LIN {X 0,Y 720.974,Z 317.138,A -85,B 0,C 180,E1 32718.045,E2 32718.045} C_VEL
LIN {X 0,Y 720.181,Z 314.525,A -85,B 0,C 180,E1 32717.982,E2 32717.982} C_VEL
LIN {X 0,Y 720.227,Z 314.61,A -85,B 0,C 180,E1 32716.261,E2 32716.261} C_VEL
LIN {X 0,Y 721.482,Z 317.961,A -85,B 0,C 180,E1 32715.916,E2 32715.916} C_VEL
LIN {X 0,Y 727.5,Z 330.946,A -85,B 0,C 180,E1 32714.519,E2 32714.519} C_VEL
LIN {X 0,Y 727.216,Z 351.094,A -85,B 0,C 180,E1 32713.184,E2 32713.184} C_VEL
LIN {X 0,Y 729.916,Z 362.068,A -85,B 0,C 180,E1 32712.841,E2 32712.841} C_VEL
LIN {X 0,Y 728.769,Z 574.456,A -85,B 0,C 180,E1 32710.185,E2 32710.185} C_VEL
LIN {X 0,Y 727.655,Z 798.892,A -85,B 0,C 180,E1 32707.472,E2 32707.472} C_VEL
LIN {X 0,Y 727.389,Z 834.661,A -85,B 0,C 180,E1 32707.008,E2 32707.008} C_VEL
LIN {X 0,Y 726.992,Z 861.421,A -85,B 0,C 180,E1 32706.503,E2 32706.503} C_VEL
LIN {X 0,Y 726.546,Z 887.78,A -85,B 0,C 180,E1 32705.847,E2 32705.847} C_VEL
LIN {X 0,Y 725.988,Z 915.933,A -85,B 0,C 180,E1 32704.967,E2 32704.967} C_VEL
LIN {X 0,Y 725.356,Z 940.667,A -85,B 0,C 180,E1 32704.031,E2 32704.031} C_VEL
LIN {X 0,Y 724.823,Z 961.723,A -85,B 0,C 180,E1 32703.11,E2 32703.11} C_VEL
LIN {X 0,Y 724.247,Z 986.24,A -85,B 0,C 180,E1 32701.889,E2 32701.889} C_VEL
LIN {X 0,Y 723.55,Z 1010.091,A -85,B 0,C 180,E1 32700.519,E2 32700.519} C_VEL
LIN {X 0,Y 723.012,Z 1029.596,A -85,B 0,C 180,E1 32699.265,E2 32699.265} C_VEL
LIN {X 0,Y 722.479,Z 1051.277,A -85,B 0,C 180,E1 32697.71,E2 32697.71} C_VEL
LIN {X 0,Y 721.914,Z 1071.822,A -85,B 0,C 180,E1 32696.043,E2 32696.043} C_VEL
LIN {X 0,Y 721.493,Z 1089.789,A -85,B 0,C 180,E1 32694.423,E2 32694.423} C_VEL
LIN {X 0,Y 721.059,Z 1108.723,A -85,B 0,C 180,E1 32692.501,E2 32692.501} C_VEL
LIN {X 0,Y 720.779,Z 1122.974,A -85,B 0,C 180,E1 32690.885,E2 32690.885} C_VEL
LIN {X 0,Y 720.524,Z 1137.042,A -85,B 0,C 180,E1 32689.116,E2 32689.116} C_VEL
LIN {X 0,Y 720.309,Z 1152.141,A -85,B 0,C 180,E1 32686.947,E2 32686.947} C_VEL
LIN {X 0,Y 720.143,Z 1162.707,A -85,B 0,C 180,E1 32685.207,E2 32685.207} C_VEL
LIN {X 0,Y 720.071,Z 1171.491,A -85,B 0,C 180,E1 32683.571,E2 32683.571} C_VEL
LIN {X 0,Y 719.987,Z 1179.518,A -85,B 0,C 180,E1 32681.86,E2 32681.86} C_VEL
LIN {X 0,Y 719.96,Z 1187.317,A -85,B 0,C 180,E1 32679.915,E2 32679.915} C_VEL
LIN {X 0,Y 719.934,Z 1194.039,A -85,B 0,C 180,E1 32677.822,E2 32677.822} C_VEL
LIN {X 0,Y 719.92,Z 1199.281,A -85,B 0,C 180,E1 32675.658,E2 32675.658} C_VEL
LIN {X 0,Y 719.915,Z 1202.793,A -85,B 0,C 180,E1 32673.503,E2 32673.503} C_VEL
LIN {X 0,Y 719.914,Z 1204.613,A -85,B 0,C 180,E1 32671.432,E2 32671.432} C_VEL
LIN {X 0,Y 719.891,Z 1204.859,A -85,B 0,C 180,E1 32669.442,E2 32669.442} C_VEL
LIN {X 0,Y 719.906,Z 1203.907,A -85,B 0,C 180,E1 32667.531,E2 32667.531} C_VEL
LIN {X 0,Y 719.907,Z 1201.173,A -85,B 0,C 180,E1 32665.379,E2 32665.379} C_VEL
LIN {X 0,Y 719.917,Z 1196.95,A -85,B 0,C 180,E1 32663.299,E2 32663.299} C_VEL
LIN {X 0,Y 719.939,Z 1191.157,A -85,B 0,C 180,E1 32661.211,E2 32661.211} C_VEL
LIN {X 0,Y 719.966,Z 1183.315,A -85,B 0,C 180,E1 32659.031,E2 32659.031} C_VEL
LIN {X 0,Y 720.059,Z 1173.533,A -85,B 0,C 180,E1 32656.836,E2 32656.836} C_VEL
LIN {X 0,Y 720.129,Z 1164.06,A -85,B 0,C 180,E1 32655.032,E2 32655.032} C_VEL
LIN {X 0,Y 720.263,Z 1154.218,A -85,B 0,C 180,E1 32653.382,E2 32653.382} C_VEL
LIN {X 0,Y 720.451,Z 1141.93,A -85,B 0,C 180,E1 32651.552,E2 32651.552} C_VEL
LIN {X 0,Y 720.732,Z 1125.799,A -85,B 0,C 180,E1 32649.451,E2 32649.451} C_VEL
LIN {X 0,Y 720.989,Z 1111.824,A -85,B 0,C 180,E1 32647.838,E2 32647.838} C_VEL
LIN {X 0,Y 721.308,Z 1097.116,A -85,B 0,C 180,E1 32646.296,E2 32646.296} C_VEL
LIN {X 0,Y 721.786,Z 1077.871,A -85,B 0,C 180,E1 32644.479,E2 32644.479} C_VEL
LIN {X 0,Y 722.256,Z 1058.515,A -85,B 0,C 180,E1 32642.86,E2 32642.86} C_VEL
LIN {X 0,Y 722.862,Z 1037.525,A -85,B 0,C 180,E1 32641.28,E2 32641.28} C_VEL
LIN {X 0,Y 723.411,Z 1014.532,A -85,B 0,C 180,E1 32639.754,E2 32639.754} C_VEL
LIN {X 0,Y 723.994,Z 993.832,A -85,B 0,C 180,E1 32638.53,E2 32638.53} C_VEL
LIN {X 0,Y 724.698,Z 969.545,A -85,B 0,C 180,E1 32637.258,E2 32637.258} C_VEL
LIN {X 0,Y 725.281,Z 944.345,A -85,B 0,C 180,E1 32636.122,E2 32636.122} C_VEL
LIN {X 0,Y 725.805,Z 921.337,A -85,B 0,C 180,E1 32635.226,E2 32635.226} C_VEL
LIN {X 0,Y 726.415,Z 895.267,A -85,B 0,C 180,E1 32634.366,E2 32634.366} C_VEL
LIN {X 0,Y 726.881,Z 868.856,A -85,B 0,C 180,E1 32633.665,E2 32633.665} C_VEL
LIN {X 0,Y 727.285,Z 842.382,A -85,B 0,C 180,E1 32633.122,E2 32633.122} C_VEL
LIN {X 0,Y 727.575,Z 814.613,A -85,B 0,C 180,E1 32632.715,E2 32632.715} C_VEL
LIN {X 0,Y 728.684,Z 590.147,A -85,B 0,C 180,E1 32630.008,E2 32630.008} C_VEL
LIN {X 0,Y 729.786,Z 383.764,A -85,B 0,C 180,E1 32627.434,E2 32627.434} C_VEL
LIN {X 0,Y 729.82,Z 346.15,A -85,B 0,C 180,E1 32626.943,E2 32626.943} C_VEL
LIN {X 0,Y 729.774,Z 330.048,A -85,B 0,C 180,E1 32626.614,E2 32626.614} C_VEL
LIN {X 0,Y 725.417,Z 323.688,A -85,B 0,C 180,E1 32626.156,E2 32626.156} C_VEL
LIN {X 0,Y 722.735,Z 319.452,A -85,B 0,C 180,E1 32625.864,E2 32625.864} C_VEL
LIN {X 0,Y 720.686,Z 316.455,A -85,B 0,C 180,E1 32625.642,E2 32625.642} C_VEL
LIN {X 0,Y 720.203,Z 314.522,A -85,B 0,C 180,E1 32625.545,E2 32625.545} C_VEL
LIN {X 0,Y 720.215,Z 314.522,A -85,B 0,C 180,E1 32622.624,E2 32622.624} C_VEL
LIN {X 0,Y 720.181,Z 314.519,A -85,B 0,C 180,E1 32619.692,E2 32619.692} C_VEL
LIN {X 0,Y 720.194,Z 314.503,A -85,B 0,C 180,E1 32616.854,E2 32616.854} C_VEL
LIN {X 0,Y 720.217,Z 314.522,A -85,B 0,C 180,E1 32613.879,E2 32613.879} C_VEL
LIN {X 0,Y 720.207,Z 314.506,A -85,B 0,C 180,E1 32610.908,E2 32610.908} C_VEL
LIN {X 0,Y 720.201,Z 314.521,A -85,B 0,C 180,E1 32607.807,E2 32607.807} C_VEL
LIN {X 0,Y 720.208,Z 314.502,A -85,B 0,C 180,E1 32604.877,E2 32604.877} C_VEL
LIN {X 0,Y 720.204,Z 314.521,A -85,B 0,C 180,E1 32601.93,E2 32601.93} C_VEL
LIN {X 0,Y 720.18,Z 314.522,A -85,B 0,C 180,E1 32599.043,E2 32599.043} C_VEL
LIN {X 0,Y 720.208,Z 314.518,A -85,B 0,C 180,E1 32596.11,E2 32596.11} C_VEL
LIN {X 0,Y 720.218,Z 314.522,A -85,B 0,C 180,E1 32593.161,E2 32593.161} C_VEL
LIN {X 0,Y 720.218,Z 314.767,A -85,B 0,C 180,E1 32591.228,E2 32591.228} C_VEL
LIN {X 0,Y 721.001,Z 318.867,A -85,B 0,C 180,E1 32591.074,E2 32591.074} C_VEL
LIN {X 0,Y 721.049,Z 390.816,A -85,B 0,C 180,E1 32588.611,E2 32588.611} C_VEL
LIN {X 0,Y 721.392,Z 472.664,A -85,B 0,C 180,E1 32585.688,E2 32585.688} C_VEL
LIN {X 0,Y 721.652,Z 538.695,A -85,B 0,C 180,E1 32583.257,E2 32583.257} C_VEL
LIN {X 0,Y 721.594,Z 602.053,A -85,B 0,C 180,E1 32580.873,E2 32580.873} C_VEL
LIN {X 0,Y 721.303,Z 676.449,A -85,B 0,C 180,E1 32578.054,E2 32578.054} C_VEL
LIN {X 0,Y 720.86,Z 755.637,A -85,B 0,C 180,E1 32575.027,E2 32575.027} C_VEL
LIN {X 0,Y 720.503,Z 836.2,A -85,B 0,C 180,E1 32571.989,E2 32571.989} C_VEL
LIN {X 0,Y 720.594,Z 839.219,A -85,B 0,C 180,E1 32571.958,E2 32571.958} C_VEL
LIN {X 0,Y 719.614,Z 846.884,A -85,B 0,C 180,E1 32571.896,E2 32571.896} C_VEL
LIN {X 0,Y 713.449,Z 867.175,A -85,B 0,C 180,E1 32571.788,E2 32571.788} C_VEL
LIN {X 0,Y 712.686,Z 873.758,A -85,B 0,C 180,E1 32571.734,E2 32571.734} C_VEL
LIN {X 0,Y 712.588,Z 952.533,A -85,B 0,C 180,E1 32570.922,E2 32570.922} C_VEL
LIN {X 0,Y 712.499,Z 966.842,A -85,B 0,C 180,E1 32570.631,E2 32570.631} C_VEL
LIN {X 0,Y 712.403,Z 980.206,A -85,B 0,C 180,E1 32570.222,E2 32570.222} C_VEL
LIN {X 0,Y 712.317,Z 993.078,A -85,B 0,C 180,E1 32569.69,E2 32569.69} C_VEL
LIN {X 0,Y 712.198,Z 1005.778,A -85,B 0,C 180,E1 32568.992,E2 32568.992} C_VEL
LIN {X 0,Y 712.115,Z 1016.953,A -85,B 0,C 180,E1 32568.212,E2 32568.212} C_VEL
LIN {X 0,Y 712.032,Z 1027.591,A -85,B 0,C 180,E1 32567.263,E2 32567.263} C_VEL
LIN {X 0,Y 711.981,Z 1035.549,A -85,B 0,C 180,E1 32566.353,E2 32566.353} C_VEL
LIN {X 0,Y 711.939,Z 1042.963,A -85,B 0,C 180,E1 32565.273,E2 32565.273} C_VEL
LIN {X 0,Y 711.925,Z 1048.677,A -85,B 0,C 180,E1 32564.105,E2 32564.105} C_VEL
LIN {X 0,Y 711.914,Z 1052.056,A -85,B 0,C 180,E1 32563.098,E2 32563.098} C_VEL
LIN {X 0,Y 711.918,Z 1054.136,A -85,B 0,C 180,E1 32562.086,E2 32562.086} C_VEL
LIN {X 0,Y 711.912,Z 1054.947,A -85,B 0,C 180,E1 32560.813,E2 32560.813} C_VEL
LIN {X 0,Y 711.918,Z 1053.936,A -85,B 0,C 180,E1 32559.701,E2 32559.701} C_VEL
LIN {X 0,Y 711.913,Z 1051.897,A -85,B 0,C 180,E1 32558.754,E2 32558.754} C_VEL
LIN {X 0,Y 711.926,Z 1048.316,A -85,B 0,C 180,E1 32557.715,E2 32557.715} C_VEL
LIN {X 0,Y 711.943,Z 1042.145,A -85,B 0,C 180,E1 32556.507,E2 32556.507} C_VEL
LIN {X 0,Y 711.982,Z 1035.188,A -85,B 0,C 180,E1 32555.511,E2 32555.511} C_VEL
LIN {X 0,Y 712.041,Z 1026.599,A -85,B 0,C 180,E1 32554.547,E2 32554.547} C_VEL
LIN {X 0,Y 712.12,Z 1016.444,A -85,B 0,C 180,E1 32553.66,E2 32553.66} C_VEL
LIN {X 0,Y 712.195,Z 1006.167,A -85,B 0,C 180,E1 32552.943,E2 32552.943} C_VEL
LIN {X 0,Y 712.308,Z 994.071,A -85,B 0,C 180,E1 32552.268,E2 32552.268} C_VEL
LIN {X 0,Y 712.4,Z 980.752,A -85,B 0,C 180,E1 32551.707,E2 32551.707} C_VEL
LIN {X 0,Y 712.484,Z 968.261,A -85,B 0,C 180,E1 32551.317,E2 32551.317} C_VEL
LIN {X 0,Y 712.585,Z 953.301,A -85,B 0,C 180,E1 32550.998,E2 32550.998} C_VEL
LIN {X 0,Y 712.639,Z 907.094,A -85,B 0,C 180,E1 32550.51,E2 32550.51} C_VEL
LIN {X 0,Y 712.62,Z 835.481,A -85,B 0,C 180,E1 32549.777,E2 32549.777} C_VEL
LIN {X 0,Y 713.066,Z 754.769,A -85,B 0,C 180,E1 32546.693,E2 32546.693} C_VEL
LIN {X 0,Y 713.49,Z 681.049,A -85,B 0,C 180,E1 32543.871,E2 32543.871} C_VEL
LIN {X 0,Y 713.925,Z 601.874,A -85,B 0,C 180,E1 32540.828,E2 32540.828} C_VEL
LIN {X 0,Y 714.318,Z 528.018,A -85,B 0,C 180,E1 32537.948,E2 32537.948} C_VEL
LIN {X 0,Y 714.295,Z 457.43,A -85,B 0,C 180,E1 32535.27,E2 32535.27} C_VEL
LIN {X 0,Y 714.435,Z 399.388,A -85,B 0,C 180,E1 32533.044,E2 32533.044} C_VEL
LIN {X 0,Y 715.772,Z 401.418,A -85,B 0,C 180,E1 32532.916,E2 32532.916} C_VEL
LIN {X 0,Y 717.784,Z 401.457,A -85,B 0,C 180,E1 32532.766,E2 32532.766} C_VEL
LIN {X 0,Y 720.642,Z 399.11,A -85,B 0,C 180,E1 32532.587,E2 32532.587} C_VEL
LIN {X 0,Y 723.62,Z 394.867,A -85,B 0,C 180,E1 32532.427,E2 32532.427} C_VEL
LIN {X 0,Y 722.239,Z 609.654,A -85,B 0,C 180,E1 32529.747,E2 32529.747} C_VEL
LIN {X 0,Y 721.025,Z 799.484,A -85,B 0,C 180,E1 32527.427,E2 32527.427} C_VEL
LIN {X 0,Y 720.629,Z 826.478,A -85,B 0,C 180,E1 32526.947,E2 32526.947} C_VEL
LIN {X 0,Y 720.054,Z 853.632,A -85,B 0,C 180,E1 32526.296,E2 32526.296} C_VEL
LIN {X 0,Y 719.485,Z 877.07,A -85,B 0,C 180,E1 32525.591,E2 32525.591} C_VEL
LIN {X 0,Y 718.87,Z 901.756,A -85,B 0,C 180,E1 32524.711,E2 32524.711} C_VEL
LIN {X 0,Y 718.073,Z 927.462,A -85,B 0,C 180,E1 32523.623,E2 32523.623} C_VEL
LIN {X 0,Y 717.352,Z 949.468,A -85,B 0,C 180,E1 32522.55,E2 32522.55} C_VEL
LIN {X 0,Y 716.647,Z 971.848,A -85,B 0,C 180,E1 32521.314,E2 32521.314} C_VEL
LIN {X 0,Y 715.878,Z 995.614,A -85,B 0,C 180,E1 32519.818,E2 32519.818} C_VEL
LIN {X 0,Y 715.153,Z 1017.098,A -85,B 0,C 180,E1 32518.293,E2 32518.293} C_VEL
LIN {X 0,Y 714.487,Z 1039.264,A -85,B 0,C 180,E1 32516.515,E2 32516.515} C_VEL
LIN {X 0,Y 713.89,Z 1057.779,A -85,B 0,C 180,E1 32514.847,E2 32514.847} C_VEL
LIN {X 0,Y 713.401,Z 1076.74,A -85,B 0,C 180,E1 32512.933,E2 32512.933} C_VEL
LIN {X 0,Y 713.009,Z 1091.871,A -85,B 0,C 180,E1 32511.212,E2 32511.212} C_VEL
LIN {X 0,Y 712.716,Z 1104.738,A -85,B 0,C 180,E1 32509.592,E2 32509.592} C_VEL
LIN {X 0,Y 712.476,Z 1116.839,A -85,B 0,C 180,E1 32507.9,E2 32507.9} C_VEL
LIN {X 0,Y 712.266,Z 1130.542,A -85,B 0,C 180,E1 32505.721,E2 32505.721} C_VEL
LIN {X 0,Y 712.109,Z 1140.422,A -85,B 0,C 180,E1 32503.894,E2 32503.894} C_VEL
LIN {X 0,Y 712.02,Z 1148.589,A -85,B 0,C 180,E1 32502.161,E2 32502.161} C_VEL
LIN {X 0,Y 711.984,Z 1156.257,A -85,B 0,C 180,E1 32500.275,E2 32500.275} C_VEL
LIN {X 0,Y 711.941,Z 1163.451,A -85,B 0,C 180,E1 32498.075,E2 32498.075} C_VEL
LIN {X 0,Y 711.921,Z 1169.015,A -85,B 0,C 180,E1 32495.805,E2 32495.805} C_VEL
LIN {X 0,Y 711.911,Z 1172.518,A -85,B 0,C 180,E1 32493.705,E2 32493.705} C_VEL
LIN {X 0,Y 711.907,Z 1174.501,A -85,B 0,C 180,E1 32491.611,E2 32491.611} C_VEL
LIN {X 0,Y 711.891,Z 1174.879,A -85,B 0,C 180,E1 32489.438,E2 32489.438} C_VEL
LIN {X 0,Y 711.906,Z 1173.876,A -85,B 0,C 180,E1 32487.425,E2 32487.425} C_VEL
LIN {X 0,Y 711.912,Z 1170.996,A -85,B 0,C 180,E1 32485.167,E2 32485.167} C_VEL
LIN {X 0,Y 711.918,Z 1166.663,A -85,B 0,C 180,E1 32483.064,E2 32483.064} C_VEL
LIN {X 0,Y 711.945,Z 1161.033,A -85,B 0,C 180,E1 32481.033,E2 32481.033} C_VEL
LIN {X 0,Y 711.994,Z 1153.18,A -85,B 0,C 180,E1 32478.827,E2 32478.827} C_VEL
LIN {X 0,Y 712.092,Z 1143.342,A -85,B 0,C 180,E1 32476.605,E2 32476.605} C_VEL
LIN {X 0,Y 712.179,Z 1134.313,A -85,B 0,C 180,E1 32474.863,E2 32474.863} C_VEL
LIN {X 0,Y 712.339,Z 1125.015,A -85,B 0,C 180,E1 32473.278,E2 32473.278} C_VEL
LIN {X 0,Y 712.524,Z 1114.561,A -85,B 0,C 180,E1 32471.68,E2 32471.68} C_VEL
LIN {X 0,Y 712.768,Z 1102.854,A -85,B 0,C 180,E1 32470.07,E2 32470.07} C_VEL
LIN {X 0,Y 713.126,Z 1087.636,A -85,B 0,C 180,E1 32468.189,E2 32468.189} C_VEL
LIN {X 0,Y 713.541,Z 1070.143,A -85,B 0,C 180,E1 32466.287,E2 32466.287} C_VEL
LIN {X 0,Y 714.064,Z 1053.157,A -85,B 0,C 180,E1 32464.63,E2 32464.63} C_VEL
LIN {X 0,Y 714.675,Z 1031.871,A -85,B 0,C 180,E1 32462.776,E2 32462.776} C_VEL
LIN {X 0,Y 715.4,Z 1010.459,A -85,B 0,C 180,E1 32461.127,E2 32461.127} C_VEL
LIN {X 0,Y 716.16,Z 985.918,A -85,B 0,C 180,E1 32459.457,E2 32459.457} C_VEL
LIN {X 0,Y 716.879,Z 964.641,A -85,B 0,C 180,E1 32458.183,E2 32458.183} C_VEL
LIN {X 0,Y 717.707,Z 940.482,A -85,B 0,C 180,E1 32456.9,E2 32456.9} C_VEL
LIN {X 0,Y 718.42,Z 915.161,A -85,B 0,C 180,E1 32455.745,E2 32455.745} C_VEL
LIN {X 0,Y 719.049,Z 892.538,A -85,B 0,C 180,E1 32454.853,E2 32454.853} C_VEL
LIN {X 0,Y 719.738,Z 867.444,A -85,B 0,C 180,E1 32454.012,E2 32454.012} C_VEL
LIN {X 0,Y 720.315,Z 841.314,A -85,B 0,C 180,E1 32453.298,E2 32453.298} C_VEL
LIN {X 0,Y 720.797,Z 815.662,A -85,B 0,C 180,E1 32452.753,E2 32452.753} C_VEL
LIN {X 0,Y 721.142,Z 789.799,A -85,B 0,C 180,E1 32452.349,E2 32452.349} C_VEL
LIN {X 0,Y 722.555,Z 560.025,A -85,B 0,C 180,E1 32449.552,E2 32449.552} C_VEL
LIN {X 0,Y 723.897,Z 350.731,A -85,B 0,C 180,E1 32446.919,E2 32446.919} C_VEL
LIN {X 0,Y 723.883,Z 335.4,A -85,B 0,C 180,E1 32446.714,E2 32446.714} C_VEL
LIN {X 0,Y 714.337,Z 320.821,A -85,B 0,C 180,E1 32445.781,E2 32445.781} C_VEL
LIN {X 0,Y 712.281,Z 315.553,A -85,B 0,C 180,E1 32445.22,E2 32445.22} C_VEL
LIN {X 0,Y 712.261,Z 315.511,A -85,B 0,C 180,E1 32442.287,E2 32442.287} C_VEL
LIN {X 0,Y 712.284,Z 315.51,A -85,B 0,C 180,E1 32439.28,E2 32439.28} C_VEL
LIN {X 0,Y 712.253,Z 315.509,A -85,B 0,C 180,E1 32436.429,E2 32436.429} C_VEL
LIN {X 0,Y 712.28,Z 315.493,A -85,B 0,C 180,E1 32433.387,E2 32433.387} C_VEL
LIN {X 0,Y 712.249,Z 315.508,A -85,B 0,C 180,E1 32430.45,E2 32430.45} C_VEL
LIN {X 0,Y 712.277,Z 315.508,A -85,B 0,C 180,E1 32427.507,E2 32427.507} C_VEL
LIN {X 0,Y 712.248,Z 315.498,A -85,B 0,C 180,E1 32424.541,E2 32424.541} C_VEL
LIN {X 0,Y 712.277,Z 315.507,A -85,B 0,C 180,E1 32421.666,E2 32421.666} C_VEL
LIN {X 0,Y 712.264,Z 315.508,A -85,B 0,C 180,E1 32418.64,E2 32418.64} C_VEL
LIN {X 0,Y 712.278,Z 315.495,A -85,B 0,C 180,E1 32415.72,E2 32415.72} C_VEL
LIN {X 0,Y 712.279,Z 315.508,A -85,B 0,C 180,E1 32412.65,E2 32412.65} C_VEL
LIN {X 0,Y 712.267,Z 315.505,A -85,B 0,C 180,E1 32409.698,E2 32409.698} C_VEL
LIN {X 0,Y 712.284,Z 315.495,A -85,B 0,C 180,E1 32406.529,E2 32406.529} C_VEL
LIN {X 0,Y 712.252,Z 315.511,A -85,B 0,C 180,E1 32403.622,E2 32403.622} C_VEL
LIN {X 0,Y 712.268,Z 315.502,A -85,B 0,C 180,E1 32400.643,E2 32400.643} C_VEL
LIN {X 0,Y 712.251,Z 315.5,A -85,B 0,C 180,E1 32397.747,E2 32397.747} C_VEL
LIN {X 0,Y 712.259,Z 315.512,A -85,B 0,C 180,E1 32394.926,E2 32394.926} C_VEL
LIN {X 0,Y 712.259,Z 315.505,A -85,B 0,C 180,E1 32392.011,E2 32392.011} C_VEL
LIN {X 0,Y 712.257,Z 315.493,A -85,B 0,C 180,E1 32389.075,E2 32389.075} C_VEL
LIN {X 0,Y 712.282,Z 315.496,A -85,B 0,C 180,E1 32386.111,E2 32386.111} C_VEL
LIN {X 0,Y 712.274,Z 315.499,A -85,B 0,C 180,E1 32383.023,E2 32383.023} C_VEL
LIN {X 0,Y 712.271,Z 315.64,A -85,B 0,C 180,E1 32381.358,E2 32381.358} C_VEL
LIN {X 0,Y 713.397,Z 318.736,A -85,B 0,C 180,E1 32380.939,E2 32380.939} C_VEL
LIN {X 0,Y 714.941,Z 320.902,A -85,B 0,C 180,E1 32380.558,E2 32380.558} C_VEL
LIN {X 0,Y 716.779,Z 324.574,A -85,B 0,C 180,E1 32380.015,E2 32380.015} C_VEL
LIN {X 0,Y 722.61,Z 335.701,A -85,B 0,C 180,E1 32378.403,E2 32378.403} C_VEL
LIN {X 0,Y 724.706,Z 339.886,A -85,B 0,C 180,E1 32377.83,E2 32377.83} C_VEL
LIN {X 0,Y 723.691,Z 373.738,A -85,B 0,C 180,E1 32375.251,E2 32375.251} C_VEL
LIN {X 0,Y 722.636,Z 410.919,A -85,B 0,C 180,E1 32372.564,E2 32372.564} C_VEL
LIN {X 0,Y 721.619,Z 447.74,A -85,B 0,C 180,E1 32370.027,E2 32370.027} C_VEL
LIN {X 0,Y 720.698,Z 486.146,A -85,B 0,C 180,E1 32367.483,E2 32367.483} C_VEL
LIN {X 0,Y 720.014,Z 532.442,A -85,B 0,C 180,E1 32364.515,E2 32364.515} C_VEL
LIN {X 0,Y 721.38,Z 542.753,A -85,B 0,C 180,E1 32363.772,E2 32363.772} C_VEL
LIN {X 0,Y 724.081,Z 551.021,A -85,B 0,C 180,E1 32363.08,E2 32363.08} C_VEL
LIN {X 0,Y 728.039,Z 557.601,A -85,B 0,C 180,E1 32362.425,E2 32362.425} C_VEL
LIN {X 0,Y 733.462,Z 562.874,A -85,B 0,C 180,E1 32361.763,E2 32361.763} C_VEL
LIN {X 0,Y 736.609,Z 564.647,A -85,B 0,C 180,E1 32361.305,E2 32361.305} C_VEL
LIN {X 0,Y 738.892,Z 564.846,A -85,B 0,C 180,E1 32360.805,E2 32360.805} C_VEL
LIN {X 0,Y 739.939,Z 563.782,A -85,B 0,C 180,E1 32360.37,E2 32360.37} C_VEL
LIN {X 0,Y 739.975,Z 561.222,A -85,B 0,C 180,E1 32359.887,E2 32359.887} C_VEL
LIN {X 0,Y 738.724,Z 557.439,A -85,B 0,C 180,E1 32359.463,E2 32359.463} C_VEL
LIN {X 0,Y 736.318,Z 552.666,A -85,B 0,C 180,E1 32359.129,E2 32359.129} C_VEL
LIN {X 0,Y 731.678,Z 544.076,A -85,B 0,C 180,E1 32358.795,E2 32358.795} C_VEL
LIN {X 0,Y 727.831,Z 533.761,A -85,B 0,C 180,E1 32358.529,E2 32358.529} C_VEL
LIN {X 0,Y 725.166,Z 522.044,A -85,B 0,C 180,E1 32358.343,E2 32358.343} C_VEL
LIN {X 0,Y 723.697,Z 508.332,A -85,B 0,C 180,E1 32358.239,E2 32358.239} C_VEL
LIN {X 0,Y 723.434,Z 499.656,A -85,B 0,C 180,E1 32358.22,E2 32358.22} C_VEL
LIN {X 0,Y 723.393,Z 331.167,A -85,B 0,C 180,E1 32358.217,E2 32358.217} C_VEL
LIN {X 0,Y 716.339,Z 322.153,A -85,B 0,C 180,E1 32357.711,E2 32357.711} C_VEL
LIN {X 0,Y 715.23,Z 320.781,A -85,B 0,C 180,E1 32357.63,E2 32357.63} C_VEL
LIN {X 0,Y 713.016,Z 317.997,A -85,B 0,C 180,E1 32357.468,E2 32357.468} C_VEL
LIN {X 0,Y 712.282,Z 315.51,A -85,B 0,C 180,E1 32357.413,E2 32357.413} C_VEL
LIN {X 0,Y 712.272,Z 315.647,A -85,B 0,C 180,E1 32356.857,E2 32356.857} C_VEL
LIN {X 0,Y 713.468,Z 318.85,A -85,B 0,C 180,E1 32356.519,E2 32356.519} C_VEL
LIN {X 0,Y 714.541,Z 321.035,A -85,B 0,C 180,E1 32356.268,E2 32356.268} C_VEL
LIN {X 0,Y 721.038,Z 335.061,A -85,B 0,C 180,E1 32354.736,E2 32354.736} C_VEL
LIN {X 0,Y 720.77,Z 351.039,A -85,B 0,C 180,E1 32353.667,E2 32353.667} C_VEL
LIN {X 0,Y 724.023,Z 364.243,A -85,B 0,C 180,E1 32353.246,E2 32353.246} C_VEL
LIN {X 0,Y 722.638,Z 575.911,A -85,B 0,C 180,E1 32350.578,E2 32350.578} C_VEL
LIN {X 0,Y 721.293,Z 799.655,A -85,B 0,C 180,E1 32347.851,E2 32347.851} C_VEL
LIN {X 0,Y 720.976,Z 834.996,A -85,B 0,C 180,E1 32347.388,E2 32347.388} C_VEL
LIN {X 0,Y 720.495,Z 862.1,A -85,B 0,C 180,E1 32346.871,E2 32346.871} C_VEL
LIN {X 0,Y 719.956,Z 888.321,A -85,B 0,C 180,E1 32346.211,E2 32346.211} C_VEL
LIN {X 0,Y 719.275,Z 916.723,A -85,B 0,C 180,E1 32345.312,E2 32345.312} C_VEL
LIN {X 0,Y 718.555,Z 940.783,A -85,B 0,C 180,E1 32344.393,E2 32344.393} C_VEL
LIN {X 0,Y 717.878,Z 962.623,A -85,B 0,C 180,E1 32343.43,E2 32343.43} C_VEL
LIN {X 0,Y 717.154,Z 987.366,A -85,B 0,C 180,E1 32342.18,E2 32342.18} C_VEL
LIN {X 0,Y 716.342,Z 1010.822,A -85,B 0,C 180,E1 32340.813,E2 32340.813} C_VEL
LIN {X 0,Y 715.668,Z 1031.083,A -85,B 0,C 180,E1 32339.492,E2 32339.492} C_VEL
LIN {X 0,Y 714.978,Z 1053.564,A -85,B 0,C 180,E1 32337.844,E2 32337.844} C_VEL
LIN {X 0,Y 714.327,Z 1073.414,A -85,B 0,C 180,E1 32336.2,E2 32336.2} C_VEL
LIN {X 0,Y 713.795,Z 1092.87,A -85,B 0,C 180,E1 32334.407,E2 32334.407} C_VEL
LIN {X 0,Y 713.307,Z 1109.504,A -85,B 0,C 180,E1 32332.672,E2 32332.672} C_VEL
LIN {X 0,Y 712.982,Z 1122.976,A -85,B 0,C 180,E1 32331.124,E2 32331.124} C_VEL
LIN {X 0,Y 712.667,Z 1137.046,A -85,B 0,C 180,E1 32329.335,E2 32329.335} C_VEL
LIN {X 0,Y 712.399,Z 1152.144,A -85,B 0,C 180,E1 32327.141,E2 32327.141} C_VEL
LIN {X 0,Y 712.202,Z 1163.143,A -85,B 0,C 180,E1 32325.303,E2 32325.303} C_VEL
LIN {X 0,Y 712.104,Z 1172.315,A -85,B 0,C 180,E1 32323.56,E2 32323.56} C_VEL
LIN {X 0,Y 712.01,Z 1180.951,A -85,B 0,C 180,E1 32321.666,E2 32321.666} C_VEL
LIN {X 0,Y 711.958,Z 1188.746,A -85,B 0,C 180,E1 32319.62,E2 32319.62} C_VEL
LIN {X 0,Y 711.929,Z 1195.357,A -85,B 0,C 180,E1 32317.423,E2 32317.423} C_VEL
LIN {X 0,Y 711.917,Z 1200.046,A -85,B 0,C 180,E1 32315.318,E2 32315.318} C_VEL
LIN {X 0,Y 711.917,Z 1203.274,A -85,B 0,C 180,E1 32313.139,E2 32313.139} C_VEL
LIN {X 0,Y 711.915,Z 1204.727,A -85,B 0,C 180,E1 32311.045,E2 32311.045} C_VEL
LIN {X 0,Y 711.895,Z 1204.816,A -85,B 0,C 180,E1 32309.275,E2 32309.275} C_VEL
LIN {X 0,Y 711.909,Z 1203.75,A -85,B 0,C 180,E1 32307.342,E2 32307.342} C_VEL
LIN {X 0,Y 711.914,Z 1200.922,A -85,B 0,C 180,E1 32305.165,E2 32305.165} C_VEL
LIN {X 0,Y 711.926,Z 1196.362,A -85,B 0,C 180,E1 32302.981,E2 32302.981} C_VEL
LIN {X 0,Y 711.949,Z 1190.352,A -85,B 0,C 180,E1 32300.868,E2 32300.868} C_VEL
LIN {X 0,Y 712.006,Z 1182.678,A -85,B 0,C 180,E1 32298.743,E2 32298.743} C_VEL
LIN {X 0,Y 712.1,Z 1173.126,A -85,B 0,C 180,E1 32296.603,E2 32296.603} C_VEL
LIN {X 0,Y 712.183,Z 1164.063,A -85,B 0,C 180,E1 32294.862,E2 32294.862} C_VEL
LIN {X 0,Y 712.366,Z 1153.699,A -85,B 0,C 180,E1 32293.108,E2 32293.108} C_VEL
LIN {X 0,Y 712.622,Z 1140.769,A -85,B 0,C 180,E1 32291.172,E2 32291.172} C_VEL
LIN {X 0,Y 712.935,Z 1125.091,A -85,B 0,C 180,E1 32289.13,E2 32289.13} C_VEL
LIN {X 0,Y 713.264,Z 1110.989,A -85,B 0,C 180,E1 32287.492,E2 32287.492} C_VEL
LIN {X 0,Y 713.71,Z 1095.411,A -85,B 0,C 180,E1 32285.852,E2 32285.852} C_VEL
LIN {X 0,Y 714.273,Z 1074.847,A -85,B 0,C 180,E1 32283.924,E2 32283.924} C_VEL
LIN {X 0,Y 714.904,Z 1055.751,A -85,B 0,C 180,E1 32282.331,E2 32282.331} C_VEL
LIN {X 0,Y 715.621,Z 1032.881,A -85,B 0,C 180,E1 32280.631,E2 32280.631} C_VEL
LIN {X 0,Y 716.283,Z 1012.242,A -85,B 0,C 180,E1 32279.275,E2 32279.275} C_VEL
LIN {X 0,Y 717.061,Z 990.171,A -85,B 0,C 180,E1 32277.975,E2 32277.975} C_VEL
LIN {X 0,Y 717.833,Z 964.661,A -85,B 0,C 180,E1 32276.666,E2 32276.666} C_VEL
LIN {X 0,Y 718.482,Z 942.857,A -85,B 0,C 180,E1 32275.692,E2 32275.692} C_VEL
LIN {X 0,Y 719.199,Z 918.806,A -85,B 0,C 180,E1 32274.762,E2 32274.762} C_VEL
LIN {X 0,Y 719.902,Z 890.448,A -85,B 0,C 180,E1 32273.849,E2 32273.849} C_VEL
LIN {X 0,Y 720.471,Z 864.075,A -85,B 0,C 180,E1 32273.173,E2 32273.173} C_VEL
LIN {X 0,Y 720.94,Z 837.046,A -85,B 0,C 180,E1 32272.646,E2 32272.646} C_VEL
LIN {X 0,Y 721.246,Z 807.217,A -85,B 0,C 180,E1 32272.24,E2 32272.24} C_VEL
LIN {X 0,Y 722.583,Z 584.166,A -85,B 0,C 180,E1 32269.524,E2 32269.524} C_VEL
LIN {X 0,Y 723.949,Z 375.621,A -85,B 0,C 180,E1 32266.9,E2 32266.9} C_VEL
LIN {X 0,Y 723.943,Z 346.826,A -85,B 0,C 180,E1 32266.515,E2 32266.515} C_VEL
LIN {X 0,Y 723.872,Z 334.141,A -85,B 0,C 180,E1 32266.255,E2 32266.255} C_VEL
LIN {X 0,Y 717.716,Z 324.946,A -85,B 0,C 180,E1 32265.59,E2 32265.59} C_VEL
LIN {X 0,Y 714.919,Z 320.514,A -85,B 0,C 180,E1 32265.275,E2 32265.275} C_VEL
LIN {X 0,Y 712.828,Z 317.584,A -85,B 0,C 180,E1 32265.046,E2 32265.046} C_VEL
LIN {X 0,Y 712.279,Z 315.508,A -85,B 0,C 180,E1 32264.949,E2 32264.949} C_VEL
LIN {X 0,Y 712.256,Z 315.513,A -85,B 0,C 180,E1 32261.822,E2 32261.822} C_VEL
LIN {X 0,Y 712.285,Z 315.51,A -85,B 0,C 180,E1 32258.865,E2 32258.865} C_VEL
LIN {X 0,Y 712.242,Z 315.495,A -85,B 0,C 180,E1 32255.901,E2 32255.901} C_VEL
LIN {X 0,Y 712.241,Z 315.51,A -85,B 0,C 180,E1 32253.196,E2 32253.196} C_VEL
LIN {X 0,Y 712.283,Z 315.497,A -85,B 0,C 180,E1 32250.148,E2 32250.148} C_VEL
LIN {X 0,Y 712.272,Z 315.504,A -85,B 0,C 180,E1 32247.235,E2 32247.235} C_VEL
LIN {X 0,Y 712.282,Z 315.498,A -85,B 0,C 180,E1 32244.152,E2 32244.152} C_VEL
LIN {X 0,Y 712.267,Z 315.509,A -85,B 0,C 180,E1 32241.062,E2 32241.062} C_VEL
LIN {X 0,Y 712.283,Z 315.505,A -85,B 0,C 180,E1 32238.074,E2 32238.074} C_VEL
LIN {X 0,Y 712.242,Z 315.511,A -85,B 0,C 180,E1 32235.015,E2 32235.015} C_VEL
LIN {X 0,Y 712.25,Z 315.512,A -85,B 0,C 180,E1 32232.239,E2 32232.239} C_VEL
LIN {X 0,Y 712.268,Z 315.656,A -85,B 0,C 180,E1 32231.37,E2 32231.37} C_VEL
LIN {X 0,Y 713.245,Z 320.296,A -85,B 0,C 180,E1 32231.196,E2 32231.196} C_VEL
LIN {X 0,Y 713.298,Z 396.474,A -85,B 0,C 180,E1 32228.586,E2 32228.586} C_VEL
LIN {X 0,Y 713.717,Z 484.597,A -85,B 0,C 180,E1 32225.426,E2 32225.426} C_VEL
LIN {X 0,Y 713.928,Z 554.263,A -85,B 0,C 180,E1 32222.85,E2 32222.85} C_VEL
LIN {X 0,Y 713.763,Z 630.95,A -85,B 0,C 180,E1 32219.96,E2 32219.96} C_VEL
LIN {X 0,Y 713.409,Z 700.395,A -85,B 0,C 180,E1 32217.309,E2 32217.309} C_VEL
LIN {X 0,Y 712.916,Z 779.916,A -85,B 0,C 180,E1 32214.253,E2 32214.253} C_VEL
LIN {X 0,Y 712.651,Z 836.618,A -85,B 0,C 180,E1 32212.108,E2 32212.108} C_VEL
LIN {X 0,Y 712.686,Z 873.758,A -85,B 0,C 180,E1 32211.734,E2 32211.734} C_VEL
LIN {X 0,Y 711.675,Z 881.423,A -85,B 0,C 180,E1 32211.672,E2 32211.672} C_VEL
LIN {X 0,Y 705.495,Z 901.707,A -85,B 0,C 180,E1 32211.561,E2 32211.561} C_VEL
LIN {X 0,Y 704.768,Z 908.287,A -85,B 0,C 180,E1 32211.506,E2 32211.506} C_VEL
LIN {X 0,Y 704.706,Z 953.239,A -85,B 0,C 180,E1 32211.026,E2 32211.026} C_VEL
LIN {X 0,Y 704.592,Z 967.916,A -85,B 0,C 180,E1 32210.71,E2 32210.71} C_VEL
LIN {X 0,Y 704.502,Z 979.281,A -85,B 0,C 180,E1 32210.359,E2 32210.359} C_VEL
LIN {X 0,Y 704.395,Z 991.495,A -85,B 0,C 180,E1 32209.862,E2 32209.862} C_VEL
LIN {X 0,Y 704.26,Z 1004.627,A -85,B 0,C 180,E1 32209.157,E2 32209.157} C_VEL
LIN {X 0,Y 704.175,Z 1014.894,A -85,B 0,C 180,E1 32208.451,E2 32208.451} C_VEL
LIN {X 0,Y 704.079,Z 1024.72,A -85,B 0,C 180,E1 32207.617,E2 32207.617} C_VEL
LIN {X 0,Y 704.004,Z 1034.007,A -85,B 0,C 180,E1 32206.614,E2 32206.614} C_VEL
LIN {X 0,Y 703.956,Z 1041.169,A -85,B 0,C 180,E1 32205.607,E2 32205.607} C_VEL
LIN {X 0,Y 703.927,Z 1047.141,A -85,B 0,C 180,E1 32204.511,E2 32204.511} C_VEL
LIN {X 0,Y 703.912,Z 1051.508,A -85,B 0,C 180,E1 32203.325,E2 32203.325} C_VEL
LIN {X 0,Y 703.917,Z 1053.809,A -85,B 0,C 180,E1 32202.303,E2 32202.303} C_VEL
LIN {X 0,Y 703.908,Z 1054.854,A -85,B 0,C 180,E1 32201.275,E2 32201.275} C_VEL
LIN {X 0,Y 703.917,Z 1054.523,A -85,B 0,C 180,E1 32200.067,E2 32200.067} C_VEL
LIN {X 0,Y 703.917,Z 1052.22,A -85,B 0,C 180,E1 32198.851,E2 32198.851} C_VEL
LIN {X 0,Y 703.926,Z 1048.943,A -85,B 0,C 180,E1 32197.84,E2 32197.84} C_VEL
LIN {X 0,Y 703.939,Z 1043.82,A -85,B 0,C 180,E1 32196.742,E2 32196.742} C_VEL
LIN {X 0,Y 703.985,Z 1036.924,A -85,B 0,C 180,E1 32195.676,E2 32195.676} C_VEL
LIN {X 0,Y 704.041,Z 1029.479,A -85,B 0,C 180,E1 32194.78,E2 32194.78} C_VEL
LIN {X 0,Y 704.122,Z 1020.201,A -85,B 0,C 180,E1 32193.882,E2 32193.882} C_VEL
LIN {X 0,Y 704.229,Z 1008.813,A -85,B 0,C 180,E1 32193.023,E2 32193.023} C_VEL
LIN {X 0,Y 704.343,Z 997.586,A -85,B 0,C 180,E1 32192.355,E2 32192.355} C_VEL
LIN {X 0,Y 704.467,Z 985.717,A -85,B 0,C 180,E1 32191.794,E2 32191.794} C_VEL
LIN {X 0,Y 704.57,Z 971.14,A -85,B 0,C 180,E1 32191.287,E2 32191.287} C_VEL
LIN {X 0,Y 704.654,Z 958.294,A -85,B 0,C 180,E1 32190.98,E2 32190.98} C_VEL
LIN {X 0,Y 704.724,Z 943.938,A -85,B 0,C 180,E1 32190.765,E2 32190.765} C_VEL
LIN {X 0,Y 704.749,Z 835.802,A -85,B 0,C 180,E1 32189.663,E2 32189.663} C_VEL
LIN {X 0,Y 705.292,Z 754.928,A -85,B 0,C 180,E1 32186.531,E2 32186.531} C_VEL
LIN {X 0,Y 705.712,Z 675.982,A -85,B 0,C 180,E1 32183.524,E2 32183.524} C_VEL
LIN {X 0,Y 706.213,Z 598.926,A -85,B 0,C 180,E1 32180.527,E2 32180.527} C_VEL
LIN {X 0,Y 706.625,Z 529.861,A -85,B 0,C 180,E1 32177.822,E2 32177.822} C_VEL
LIN {X 0,Y 706.718,Z 457.885,A -85,B 0,C 180,E1 32175.058,E2 32175.058} C_VEL
LIN {X 0,Y 706.775,Z 415.254,A -85,B 0,C 180,E1 32173.409,E2 32173.409} C_VEL
LIN {X 0,Y 708.063,Z 417.224,A -85,B 0,C 180,E1 32173.284,E2 32173.284} C_VEL
LIN {X 0,Y 709.871,Z 417.364,A -85,B 0,C 180,E1 32173.144,E2 32173.144} C_VEL
LIN {X 0,Y 712.699,Z 415.211,A -85,B 0,C 180,E1 32172.96,E2 32172.96} C_VEL
LIN {X 0,Y 716.31,Z 409.789,A -85,B 0,C 180,E1 32172.764,E2 32172.764} C_VEL
LIN {X 0,Y 717.577,Z 409.589,A -85,B 0,C 180,E1 32172.673,E2 32172.673} C_VEL
LIN {X 0,Y 716.004,Z 620.642,A -85,B 0,C 180,E1 32170.023,E2 32170.023} C_VEL
LIN {X 0,Y 714.66,Z 799.521,A -85,B 0,C 180,E1 32167.819,E2 32167.819} C_VEL
LIN {X 0,Y 714.194,Z 826.514,A -85,B 0,C 180,E1 32167.336,E2 32167.336} C_VEL
LIN {X 0,Y 713.526,Z 853.637,A -85,B 0,C 180,E1 32166.682,E2 32166.682} C_VEL
LIN {X 0,Y 712.863,Z 876.436,A -85,B 0,C 180,E1 32165.995,E2 32165.995} C_VEL
LIN {X 0,Y 712.155,Z 900.241,A -85,B 0,C 180,E1 32165.146,E2 32165.146} C_VEL
LIN {X 0,Y 711.296,Z 925.704,A -85,B 0,C 180,E1 32164.074,E2 32164.074} C_VEL
LIN {X 0,Y 710.414,Z 948.595,A -85,B 0,C 180,E1 32162.956,E2 32162.956} C_VEL
LIN {X 0,Y 709.572,Z 970.293,A -85,B 0,C 180,E1 32161.757,E2 32161.757} C_VEL
LIN {X 0,Y 708.659,Z 994.966,A -85,B 0,C 180,E1 32160.2,E2 32160.2} C_VEL
LIN {X 0,Y 707.824,Z 1016.123,A -85,B 0,C 180,E1 32158.688,E2 32158.688} C_VEL
LIN {X 0,Y 707.005,Z 1038.259,A -85,B 0,C 180,E1 32156.909,E2 32156.909} C_VEL
LIN {X 0,Y 706.312,Z 1057.323,A -85,B 0,C 180,E1 32155.177,E2 32155.177} C_VEL
LIN {X 0,Y 705.724,Z 1075.95,A -85,B 0,C 180,E1 32153.285,E2 32153.285} C_VEL
LIN {X 0,Y 705.224,Z 1091.877,A -85,B 0,C 180,E1 32151.458,E2 32151.458} C_VEL
LIN {X 0,Y 704.88,Z 1104.743,A -85,B 0,C 180,E1 32149.818,E2 32149.818} C_VEL
LIN {X 0,Y 704.577,Z 1117.425,A -85,B 0,C 180,E1 32148.022,E2 32148.022} C_VEL
LIN {X 0,Y 704.324,Z 1131.01,A -85,B 0,C 180,E1 32145.818,E2 32145.818} C_VEL
LIN {X 0,Y 704.149,Z 1140.836,A -85,B 0,C 180,E1 32143.97,E2 32143.97} C_VEL
LIN {X 0,Y 704.053,Z 1148.654,A -85,B 0,C 180,E1 32142.286,E2 32142.286} C_VEL
LIN {X 0,Y 703.993,Z 1156.256,A -85,B 0,C 180,E1 32140.393,E2 32140.393} C_VEL
LIN {X 0,Y 703.949,Z 1163.207,A -85,B 0,C 180,E1 32138.249,E2 32138.249} C_VEL
LIN {X 0,Y 703.924,Z 1168.674,A -85,B 0,C 180,E1 32136.035,E2 32136.035} C_VEL
LIN {X 0,Y 703.912,Z 1172.313,A -85,B 0,C 180,E1 32133.911,E2 32133.911} C_VEL
LIN {X 0,Y 703.907,Z 1174.45,A -85,B 0,C 180,E1 32131.71,E2 32131.71} C_VEL
LIN {X 0,Y 703.89,Z 1174.904,A -85,B 0,C 180,E1 32129.513,E2 32129.513} C_VEL
LIN {X 0,Y 703.905,Z 1173.954,A -85,B 0,C 180,E1 32127.477,E2 32127.477} C_VEL
LIN {X 0,Y 703.911,Z 1171.129,A -85,B 0,C 180,E1 32125.194,E2 32125.194} C_VEL
LIN {X 0,Y 703.921,Z 1166.855,A -85,B 0,C 180,E1 32123.066,E2 32123.066} C_VEL
LIN {X 0,Y 703.951,Z 1161.276,A -85,B 0,C 180,E1 32121.012,E2 32121.012} C_VEL
LIN {X 0,Y 704.002,Z 1153.816,A -85,B 0,C 180,E1 32118.864,E2 32118.864} C_VEL
LIN {X 0,Y 704.127,Z 1143.75,A -85,B 0,C 180,E1 32116.534,E2 32116.534} C_VEL
LIN {X 0,Y 704.233,Z 1134.776,A -85,B 0,C 180,E1 32114.773,E2 32114.773} C_VEL
LIN {X 0,Y 704.435,Z 1124.963,A -85,B 0,C 180,E1 32113.077,E2 32113.077} C_VEL
LIN {X 0,Y 704.655,Z 1114.557,A -85,B 0,C 180,E1 32111.468,E2 32111.468} C_VEL
LIN {X 0,Y 704.935,Z 1102.851,A -85,B 0,C 180,E1 32109.839,E2 32109.839} C_VEL
LIN {X 0,Y 705.369,Z 1087.629,A -85,B 0,C 180,E1 32107.937,E2 32107.937} C_VEL
LIN {X 0,Y 705.875,Z 1070.14,A -85,B 0,C 180,E1 32106.014,E2 32106.014} C_VEL
LIN {X 0,Y 706.475,Z 1053.155,A -85,B 0,C 180,E1 32104.338,E2 32104.338} C_VEL
LIN {X 0,Y 707.23,Z 1031.869,A -85,B 0,C 180,E1 32102.465,E2 32102.465} C_VEL
LIN {X 0,Y 708.072,Z 1009.851,A -85,B 0,C 180,E1 32100.753,E2 32100.753} C_VEL
LIN {X 0,Y 708.972,Z 985.915,A -85,B 0,C 180,E1 32099.114,E2 32099.114} C_VEL
LIN {X 0,Y 709.818,Z 964.637,A -85,B 0,C 180,E1 32097.829,E2 32097.829} C_VEL
LIN {X 0,Y 710.766,Z 940.462,A -85,B 0,C 180,E1 32096.535,E2 32096.535} C_VEL
LIN {X 0,Y 711.618,Z 915.041,A -85,B 0,C 180,E1 32095.366,E2 32095.366} C_VEL
LIN {X 0,Y 712.37,Z 892.528,A -85,B 0,C 180,E1 32094.474,E2 32094.474} C_VEL
LIN {X 0,Y 713.155,Z 867.431,A -85,B 0,C 180,E1 32093.627,E2 32093.627} C_VEL
LIN {X 0,Y 713.843,Z 841.039,A -85,B 0,C 180,E1 32092.904,E2 32092.904} C_VEL
LIN {X 0,Y 714.387,Z 815.682,A -85,B 0,C 180,E1 32092.363,E2 32092.363} C_VEL
LIN {X 0,Y 714.793,Z 789.949,A -85,B 0,C 180,E1 32091.958,E2 32091.958} C_VEL
LIN {X 0,Y 716.448,Z 560.834,A -85,B 0,C 180,E1 32089.146,E2 32089.146} C_VEL
LIN {X 0,Y 718.032,Z 351.549,A -85,B 0,C 180,E1 32086.492,E2 32086.492} C_VEL
LIN {X 0,Y 717.949,Z 338.826,A -85,B 0,C 180,E1 32086.314,E2 32086.314} C_VEL
LIN {X 0,Y 706.118,Z 320.857,A -85,B 0,C 180,E1 32085.132,E2 32085.132} C_VEL
LIN {X 0,Y 704.347,Z 316.72,A -85,B 0,C 180,E1 32084.668,E2 32084.668} C_VEL
LIN {X 0,Y 704.335,Z 316.499,A -85,B 0,C 180,E1 32081.818,E2 32081.818} C_VEL
LIN {X 0,Y 704.324,Z 316.5,A -85,B 0,C 180,E1 32078.928,E2 32078.928} C_VEL
LIN {X 0,Y 704.312,Z 316.498,A -85,B 0,C 180,E1 32076.098,E2 32076.098} C_VEL
LIN {X 0,Y 704.334,Z 316.481,A -85,B 0,C 180,E1 32073.228,E2 32073.228} C_VEL
LIN {X 0,Y 704.313,Z 316.495,A -85,B 0,C 180,E1 32070.264,E2 32070.264} C_VEL
LIN {X 0,Y 704.347,Z 316.499,A -85,B 0,C 180,E1 32067.297,E2 32067.297} C_VEL
LIN {X 0,Y 704.319,Z 316.486,A -85,B 0,C 180,E1 32064.223,E2 32064.223} C_VEL
LIN {X 0,Y 704.342,Z 316.49,A -85,B 0,C 180,E1 32061.31,E2 32061.31} C_VEL
LIN {X 0,Y 704.336,Z 316.498,A -85,B 0,C 180,E1 32058.199,E2 32058.199} C_VEL
LIN {X 0,Y 704.331,Z 316.483,A -85,B 0,C 180,E1 32055.226,E2 32055.226} C_VEL
LIN {X 0,Y 704.338,Z 316.493,A -85,B 0,C 180,E1 32052.212,E2 32052.212} C_VEL
LIN {X 0,Y 704.313,Z 316.498,A -85,B 0,C 180,E1 32049.314,E2 32049.314} C_VEL
LIN {X 0,Y 704.34,Z 316.481,A -85,B 0,C 180,E1 32046.357,E2 32046.357} C_VEL
LIN {X 0,Y 704.31,Z 316.5,A -85,B 0,C 180,E1 32043.418,E2 32043.418} C_VEL
LIN {X 0,Y 704.341,Z 316.49,A -85,B 0,C 180,E1 32040.488,E2 32040.488} C_VEL
LIN {X 0,Y 704.309,Z 316.485,A -85,B 0,C 180,E1 32037.478,E2 32037.478} C_VEL
LIN {X 0,Y 704.345,Z 316.494,A -85,B 0,C 180,E1 32034.542,E2 32034.542} C_VEL
LIN {X 0,Y 704.32,Z 316.498,A -85,B 0,C 180,E1 32031.427,E2 32031.427} C_VEL
LIN {X 0,Y 704.338,Z 316.48,A -85,B 0,C 180,E1 32028.536,E2 32028.536} C_VEL
LIN {X 0,Y 704.338,Z 316.474,A -85,B 0,C 180,E1 32025.363,E2 32025.363} C_VEL
LIN {X 0,Y 704.323,Z 316.474,A -85,B 0,C 180,E1 32022.399,E2 32022.399} C_VEL
LIN {X 0,Y 704.365,Z 316.746,A -85,B 0,C 180,E1 32022.268,E2 32022.268} C_VEL
LIN {X 0,Y 705.824,Z 320.21,A -85,B 0,C 180,E1 32021.755,E2 32021.755} C_VEL
LIN {X 0,Y 707.019,Z 321.916,A -85,B 0,C 180,E1 32021.446,E2 32021.446} C_VEL
LIN {X 0,Y 708.795,Z 325.516,A -85,B 0,C 180,E1 32020.896,E2 32020.896} C_VEL
LIN {X 0,Y 709.884,Z 327.497,A -85,B 0,C 180,E1 32020.585,E2 32020.585} C_VEL
LIN {X 0,Y 712.587,Z 332.638,A -85,B 0,C 180,E1 32019.807,E2 32019.807} C_VEL
LIN {X 0,Y 718.888,Z 344.57,A -85,B 0,C 180,E1 32018.077,E2 32018.077} C_VEL
LIN {X 0,Y 717.683,Z 378.598,A -85,B 0,C 180,E1 32015.469,E2 32015.469} C_VEL
LIN {X 0,Y 716.458,Z 415.255,A -85,B 0,C 180,E1 32012.802,E2 32012.802} C_VEL
LIN {X 0,Y 715.273,Z 452.087,A -85,B 0,C 180,E1 32010.247,E2 32010.247} C_VEL
LIN {X 0,Y 714.178,Z 490.739,A -85,B 0,C 180,E1 32007.668,E2 32007.668} C_VEL
LIN {X 0,Y 713.342,Z 535.088,A -85,B 0,C 180,E1 32004.801,E2 32004.801} C_VEL
LIN {X 0,Y 714.668,Z 545.999,A -85,B 0,C 180,E1 32004.011,E2 32004.011} C_VEL
LIN {X 0,Y 717.469,Z 555.035,A -85,B 0,C 180,E1 32003.255,E2 32003.255} C_VEL
LIN {X 0,Y 721.639,Z 562.32,A -85,B 0,C 180,E1 32002.535,E2 32002.535} C_VEL
LIN {X 0,Y 726.976,Z 567.923,A -85,B 0,C 180,E1 32001.862,E2 32001.862} C_VEL
LIN {X 0,Y 730.996,Z 570.707,A -85,B 0,C 180,E1 32001.41,E2 32001.41} C_VEL
LIN {X 0,Y 734.129,Z 571.797,A -85,B 0,C 180,E1 32000.924,E2 32000.924} C_VEL
LIN {X 0,Y 736.105,Z 571.355,A -85,B 0,C 180,E1 32000.426,E2 32000.426} C_VEL
LIN {X 0,Y 736.853,Z 569.556,A -85,B 0,C 180,E1 31999.934,E2 31999.934} C_VEL
LIN {X 0,Y 736.275,Z 566.387,A -85,B 0,C 180,E1 31999.461,E2 31999.461} C_VEL
LIN {X 0,Y 734.382,Z 562.168,A -85,B 0,C 180,E1 31999.065,E2 31999.065} C_VEL
LIN {X 0,Y 731.35,Z 557.084,A -85,B 0,C 180,E1 31998.772,E2 31998.772} C_VEL
LIN {X 0,Y 726.241,Z 547.547,A -85,B 0,C 180,E1 31998.418,E2 31998.418} C_VEL
LIN {X 0,Y 722.183,Z 536.4,A -85,B 0,C 180,E1 31998.132,E2 31998.132} C_VEL
LIN {X 0,Y 719.395,Z 524.056,A -85,B 0,C 180,E1 31997.932,E2 31997.932} C_VEL
LIN {X 0,Y 717.819,Z 509.85,A -85,B 0,C 180,E1 31997.819,E2 31997.819} C_VEL
LIN {X 0,Y 717.489,Z 499.787,A -85,B 0,C 180,E1 31997.795,E2 31997.795} C_VEL
LIN {X 0,Y 717.356,Z 334.772,A -85,B 0,C 180,E1 31997.785,E2 31997.785} C_VEL
LIN {X 0,Y 710.809,Z 326.355,A -85,B 0,C 180,E1 31997.305,E2 31997.305} C_VEL
LIN {X 0,Y 707.691,Z 322.076,A -85,B 0,C 180,E1 31997.071,E2 31997.071} C_VEL
LIN {X 0,Y 706.332,Z 321.169,A -85,B 0,C 180,E1 31996.959,E2 31996.959} C_VEL
LIN {X 0,Y 714.556,Z 339.147,A -85,B 0,C 180,E1 31994.961,E2 31994.961} C_VEL
LIN {X 0,Y 714.39,Z 351.16,A -85,B 0,C 180,E1 31994.156,E2 31994.156} C_VEL
LIN {X 0,Y 718.166,Z 366.415,A -85,B 0,C 180,E1 31993.657,E2 31993.657} C_VEL
LIN {X 0,Y 716.54,Z 577.523,A -85,B 0,C 180,E1 31990.976,E2 31990.976} C_VEL
LIN {X 0,Y 714.959,Z 801.131,A -85,B 0,C 180,E1 31988.228,E2 31988.228} C_VEL
LIN {X 0,Y 714.592,Z 835.485,A -85,B 0,C 180,E1 31987.772,E2 31987.772} C_VEL
LIN {X 0,Y 714.026,Z 862.916,A -85,B 0,C 180,E1 31987.242,E2 31987.242} C_VEL
LIN {X 0,Y 713.392,Z 889.053,A -85,B 0,C 180,E1 31986.576,E2 31986.576} C_VEL
LIN {X 0,Y 712.631,Z 916.26,A -85,B 0,C 180,E1 31985.708,E2 31985.708} C_VEL
LIN {X 0,Y 711.794,Z 940.685,A -85,B 0,C 180,E1 31984.771,E2 31984.771} C_VEL
LIN {X 0,Y 710.981,Z 962.941,A -85,B 0,C 180,E1 31983.782,E2 31983.782} C_VEL
LIN {X 0,Y 710.088,Z 988.203,A -85,B 0,C 180,E1 31982.492,E2 31982.492} C_VEL
LIN {X 0,Y 709.178,Z 1010.992,A -85,B 0,C 180,E1 31981.148,E2 31981.148} C_VEL
LIN {X 0,Y 708.397,Z 1030.932,A -85,B 0,C 180,E1 31979.836,E2 31979.836} C_VEL
LIN {X 0,Y 707.548,Z 1053.569,A -85,B 0,C 180,E1 31978.163,E2 31978.163} C_VEL
LIN {X 0,Y 706.795,Z 1073.861,A -85,B 0,C 180,E1 31976.462,E2 31976.462} C_VEL
LIN {X 0,Y 706.12,Z 1093.552,A -85,B 0,C 180,E1 31974.619,E2 31974.619} C_VEL
LIN {X 0,Y 705.562,Z 1110.284,A -85,B 0,C 180,E1 31972.847,E2 31972.847} C_VEL
LIN {X 0,Y 705.158,Z 1124.399,A -85,B 0,C 180,E1 31971.196,E2 31971.196} C_VEL
LIN {X 0,Y 704.76,Z 1140.336,A -85,B 0,C 180,E1 31969.108,E2 31969.108} C_VEL
LIN {X 0,Y 704.464,Z 1153.715,A -85,B 0,C 180,E1 31967.085,E2 31967.085} C_VEL
LIN {X 0,Y 704.248,Z 1164.076,A -85,B 0,C 180,E1 31965.311,E2 31965.311} C_VEL
LIN {X 0,Y 704.128,Z 1173.96,A -85,B 0,C 180,E1 31963.382,E2 31963.382} C_VEL
LIN {X 0,Y 703.991,Z 1184.281,A -85,B 0,C 180,E1 31960.97,E2 31960.97} C_VEL
LIN {X 0,Y 703.949,Z 1191.411,A -85,B 0,C 180,E1 31958.905,E2 31958.905} C_VEL
LIN {X 0,Y 703.921,Z 1197.343,A -85,B 0,C 180,E1 31956.688,E2 31956.688} C_VEL
LIN {X 0,Y 703.909,Z 1201.424,A -85,B 0,C 180,E1 31954.561,E2 31954.561} C_VEL
LIN {X 0,Y 703.907,Z 1203.985,A -85,B 0,C 180,E1 31952.441,E2 31952.441} C_VEL
LIN {X 0,Y 703.898,Z 1204.951,A -85,B 0,C 180,E1 31950.243,E2 31950.243} C_VEL
LIN {X 0,Y 703.913,Z 1204.209,A -85,B 0,C 180,E1 31947.882,E2 31947.882} C_VEL
LIN {X 0,Y 703.918,Z 1201.92,A -85,B 0,C 180,E1 31945.763,E2 31945.763} C_VEL
LIN {X 0,Y 703.927,Z 1197.908,A -85,B 0,C 180,E1 31943.556,E2 31943.556} C_VEL
LIN {X 0,Y 703.951,Z 1192.381,A -85,B 0,C 180,E1 31941.422,E2 31941.422} C_VEL
LIN {X 0,Y 703.982,Z 1185.221,A -85,B 0,C 180,E1 31939.276,E2 31939.276} C_VEL
LIN {X 0,Y 704.11,Z 1175.93,A -85,B 0,C 180,E1 31937.033,E2 31937.033} C_VEL
LIN {X 0,Y 704.228,Z 1165.273,A -85,B 0,C 180,E1 31934.905,E2 31934.905} C_VEL
LIN {X 0,Y 704.437,Z 1154.707,A -85,B 0,C 180,E1 31933.076,E2 31933.076} C_VEL
LIN {X 0,Y 704.708,Z 1142.52,A -85,B 0,C 180,E1 31931.21,E2 31931.21} C_VEL
LIN {X 0,Y 705.106,Z 1126.514,A -85,B 0,C 180,E1 31929.062,E2 31929.062} C_VEL
LIN {X 0,Y 705.514,Z 1111.732,A -85,B 0,C 180,E1 31927.314,E2 31927.314} C_VEL
LIN {X 0,Y 706.031,Z 1096.267,A -85,B 0,C 180,E1 31925.661,E2 31925.661} C_VEL
LIN {X 0,Y 706.709,Z 1075.867,A -85,B 0,C 180,E1 31923.714,E2 31923.714} C_VEL
LIN {X 0,Y 707.427,Z 1056.863,A -85,B 0,C 180,E1 31922.105,E2 31922.105} C_VEL
LIN {X 0,Y 708.271,Z 1034.598,A -85,B 0,C 180,E1 31920.416,E2 31920.416} C_VEL
LIN {X 0,Y 709.089,Z 1012.972,A -85,B 0,C 180,E1 31918.976,E2 31918.976} C_VEL
LIN {X 0,Y 709.923,Z 992.24,A -85,B 0,C 180,E1 31917.737,E2 31917.737} C_VEL
LIN {X 0,Y 710.852,Z 967.646,A -85,B 0,C 180,E1 31916.44,E2 31916.44} C_VEL
LIN {X 0,Y 711.659,Z 943.985,A -85,B 0,C 180,E1 31915.366,E2 31915.366} C_VEL
LIN {X 0,Y 712.482,Z 920.09,A -85,B 0,C 180,E1 31914.429,E2 31914.429} C_VEL
LIN {X 0,Y 713.299,Z 892.406,A -85,B 0,C 180,E1 31913.52,E2 31913.52} C_VEL
LIN {X 0,Y 713.991,Z 865.377,A -85,B 0,C 180,E1 31912.812,E2 31912.812} C_VEL
LIN {X 0,Y 714.525,Z 838.594,A -85,B 0,C 180,E1 31912.28,E2 31912.28} C_VEL
LIN {X 0,Y 714.896,Z 809.889,A -85,B 0,C 180,E1 31911.878,E2 31911.878} C_VEL
LIN {X 0,Y 716.467,Z 587.05,A -85,B 0,C 180,E1 31909.143,E2 31909.143} C_VEL
LIN {X 0,Y 718.057,Z 379.972,A -85,B 0,C 180,E1 31906.518,E2 31906.518} C_VEL
LIN {X 0,Y 718.125,Z 348.062,A -85,B 0,C 180,E1 31906.09,E2 31906.09} C_VEL
LIN {X 0,Y 717.963,Z 338.017,A -85,B 0,C 180,E1 31905.884,E2 31905.884} C_VEL
LIN {X 0,Y 709.931,Z 326.045,A -85,B 0,C 180,E1 31904.994,E2 31904.994} C_VEL
LIN {X 0,Y 707.011,Z 321.525,A -85,B 0,C 180,E1 31904.659,E2 31904.659} C_VEL
LIN {X 0,Y 704.871,Z 318.535,A -85,B 0,C 180,E1 31904.417,E2 31904.417} C_VEL
LIN {X 0,Y 704.339,Z 316.499,A -85,B 0,C 180,E1 31904.316,E2 31904.316} C_VEL
LIN {X 0,Y 704.338,Z 316.619,A -85,B 0,C 180,E1 31902.998,E2 31902.998} C_VEL
LIN {X 0,Y 705.069,Z 318.982,A -85,B 0,C 180,E1 31902.824,E2 31902.824} C_VEL
LIN {X 0,Y 706.122,Z 320.639,A -85,B 0,C 180,E1 31902.459,E2 31902.459} C_VEL
LIN {X 0,Y 706.44,Z 321.011,A -85,B 0,C 180,E1 31902.005,E2 31902.005} C_VEL
LIN {X 0,Y 705.699,Z 320.059,A -85,B 0,C 180,E1 31901.537,E2 31901.537} C_VEL
LIN {X 0,Y 704.616,Z 317.837,A -85,B 0,C 180,E1 31901.199,E2 31901.199} C_VEL
LIN {X 0,Y 704.327,Z 316.487,A -85,B 0,C 180,E1 31901.076,E2 31901.076} C_VEL
LIN {X 0,Y 704.327,Z 316.491,A -85,B 0,C 180,E1 31897.931,E2 31897.931} C_VEL
LIN {X 0,Y 704.339,Z 316.49,A -85,B 0,C 180,E1 31894.997,E2 31894.997} C_VEL
LIN {X 0,Y 704.31,Z 316.479,A -85,B 0,C 180,E1 31891.974,E2 31891.974} C_VEL
LIN {X 0,Y 704.305,Z 316.5,A -85,B 0,C 180,E1 31889.141,E2 31889.141} C_VEL
LIN {X 0,Y 704.341,Z 316.474,A -85,B 0,C 180,E1 31886.2,E2 31886.2} C_VEL
LIN {X 0,Y 704.321,Z 316.499,A -85,B 0,C 180,E1 31883.245,E2 31883.245} C_VEL
LIN {X 0,Y 704.337,Z 316.491,A -85,B 0,C 180,E1 31880.22,E2 31880.22} C_VEL
LIN {X 0,Y 704.336,Z 316.493,A -85,B 0,C 180,E1 31877.174,E2 31877.174} C_VEL
LIN {X 0,Y 704.341,Z 316.497,A -85,B 0,C 180,E1 31874.165,E2 31874.165} C_VEL
LIN {X 0,Y 704.326,Z 316.571,A -85,B 0,C 180,E1 31871.519,E2 31871.519} C_VEL
LIN {X 0,Y 705.487,Z 321.677,A -85,B 0,C 180,E1 31871.321,E2 31871.321} C_VEL
LIN {X 0,Y 705.549,Z 396.393,A -85,B 0,C 180,E1 31868.763,E2 31868.763} C_VEL
LIN {X 0,Y 705.909,Z 478.74,A -85,B 0,C 180,E1 31865.813,E2 31865.813} C_VEL
LIN {X 0,Y 706.145,Z 540.661,A -85,B 0,C 180,E1 31863.531,E2 31863.531} C_VEL
LIN {X 0,Y 706.081,Z 605.396,A -85,B 0,C 180,E1 31861.095,E2 31861.095} C_VEL
LIN {X 0,Y 705.723,Z 687.618,A -85,B 0,C 180,E1 31857.97,E2 31857.97} C_VEL
LIN {X 0,Y 705.217,Z 765.885,A -85,B 0,C 180,E1 31854.957,E2 31854.957} C_VEL
LIN {X 0,Y 704.777,Z 836.544,A -85,B 0,C 180,E1 31852.235,E2 31852.235} C_VEL
LIN {X 0,Y 704.768,Z 908.287,A -85,B 0,C 180,E1 31851.506,E2 31851.506} C_VEL
LIN {X 0,Y 703.793,Z 915.952,A -85,B 0,C 180,E1 31851.443,E2 31851.443} C_VEL
LIN {X 0,Y 697.592,Z 936.234,A -85,B 0,C 180,E1 31851.328,E2 31851.328} C_VEL
LIN {X 0,Y 696.848,Z 942.817,A -85,B 0,C 180,E1 31851.27,E2 31851.27} C_VEL
LIN {X 0,Y 696.778,Z 957.841,A -85,B 0,C 180,E1 31851.054,E2 31851.054} C_VEL
LIN {X 0,Y 696.685,Z 969.88,A -85,B 0,C 180,E1 31850.771,E2 31850.771} C_VEL
LIN {X 0,Y 696.581,Z 983.128,A -85,B 0,C 180,E1 31850.332,E2 31850.332} C_VEL
LIN {X 0,Y 696.428,Z 996.558,A -85,B 0,C 180,E1 31849.712,E2 31849.712} C_VEL
LIN {X 0,Y 696.291,Z 1007.341,A -85,B 0,C 180,E1 31849.073,E2 31849.073} C_VEL
LIN {X 0,Y 696.184,Z 1017.726,A -85,B 0,C 180,E1 31848.316,E2 31848.316} C_VEL
LIN {X 0,Y 696.073,Z 1027.759,A -85,B 0,C 180,E1 31847.388,E2 31847.388} C_VEL
LIN {X 0,Y 696.009,Z 1035.037,A -85,B 0,C 180,E1 31846.542,E2 31846.542} C_VEL
LIN {X 0,Y 695.961,Z 1041.486,A -85,B 0,C 180,E1 31845.608,E2 31845.608} C_VEL
LIN {X 0,Y 695.928,Z 1047.387,A -85,B 0,C 180,E1 31844.5,E2 31844.5} C_VEL
LIN {X 0,Y 695.912,Z 1051.645,A -85,B 0,C 180,E1 31843.3,E2 31843.3} C_VEL
LIN {X 0,Y 695.917,Z 1053.892,A -85,B 0,C 180,E1 31842.266,E2 31842.266} C_VEL
LIN {X 0,Y 695.909,Z 1054.881,A -85,B 0,C 180,E1 31841.225,E2 31841.225} C_VEL
LIN {X 0,Y 695.918,Z 1054.444,A -85,B 0,C 180,E1 31839.995,E2 31839.995} C_VEL
LIN {X 0,Y 695.917,Z 1052.213,A -85,B 0,C 180,E1 31838.825,E2 31838.825} C_VEL
LIN {X 0,Y 695.928,Z 1048.914,A -85,B 0,C 180,E1 31837.798,E2 31837.798} C_VEL
LIN {X 0,Y 695.945,Z 1043.586,A -85,B 0,C 180,E1 31836.647,E2 31836.647} C_VEL
LIN {X 0,Y 695.999,Z 1036.49,A -85,B 0,C 180,E1 31835.559,E2 31835.559} C_VEL
LIN {X 0,Y 696.065,Z 1028.966,A -85,B 0,C 180,E1 31834.654,E2 31834.654} C_VEL
LIN {X 0,Y 696.162,Z 1019.566,A -85,B 0,C 180,E1 31833.744,E2 31833.744} C_VEL
LIN {X 0,Y 696.283,Z 1008.575,A -85,B 0,C 180,E1 31832.917,E2 31832.917} C_VEL
LIN {X 0,Y 696.409,Z 997.978,A -85,B 0,C 180,E1 31832.277,E2 31832.277} C_VEL
LIN {X 0,Y 696.534,Z 987.618,A -85,B 0,C 180,E1 31831.77,E2 31831.77} C_VEL
LIN {X 0,Y 696.671,Z 974.207,A -85,B 0,C 180,E1 31831.262,E2 31831.262} C_VEL
LIN {X 0,Y 696.769,Z 959.771,A -85,B 0,C 180,E1 31830.894,E2 31830.894} C_VEL
LIN {X 0,Y 696.842,Z 945.641,A -85,B 0,C 180,E1 31830.669,E2 31830.669} C_VEL
LIN {X 0,Y 696.904,Z 835.953,A -85,B 0,C 180,E1 31829.528,E2 31829.528} C_VEL
LIN {X 0,Y 697.519,Z 755.812,A -85,B 0,C 180,E1 31826.394,E2 31826.394} C_VEL
LIN {X 0,Y 697.999,Z 676.196,A -85,B 0,C 180,E1 31823.342,E2 31823.342} C_VEL
LIN {X 0,Y 698.499,Z 599.74,A -85,B 0,C 180,E1 31820.367,E2 31820.367} C_VEL
LIN {X 0,Y 698.881,Z 542.449,A -85,B 0,C 180,E1 31818.116,E2 31818.116} C_VEL
LIN {X 0,Y 699.09,Z 477.257,A -85,B 0,C 180,E1 31815.579,E2 31815.579} C_VEL
LIN {X 0,Y 699.169,Z 431.009,A -85,B 0,C 180,E1 31813.783,E2 31813.783} C_VEL
LIN {X 0,Y 700.389,Z 432.953,A -85,B 0,C 180,E1 31813.66,E2 31813.66} C_VEL
LIN {X 0,Y 701.996,Z 433.21,A -85,B 0,C 180,E1 31813.531,E2 31813.531} C_VEL
LIN {X 0,Y 704.689,Z 431.388,A -85,B 0,C 180,E1 31813.348,E2 31813.348} C_VEL
LIN {X 0,Y 708.201,Z 426.408,A -85,B 0,C 180,E1 31813.148,E2 31813.148} C_VEL
LIN {X 0,Y 708.829,Z 425.434,A -85,B 0,C 180,E1 31813.114,E2 31813.114} C_VEL
LIN {X 0,Y 711.542,Z 424.915,A -85,B 0,C 180,E1 31812.916,E2 31812.916} C_VEL
LIN {X 0,Y 709.783,Z 631.938,A -85,B 0,C 180,E1 31810.299,E2 31810.299} C_VEL
LIN {X 0,Y 708.33,Z 799.428,A -85,B 0,C 180,E1 31808.219,E2 31808.219} C_VEL
LIN {X 0,Y 707.791,Z 826.572,A -85,B 0,C 180,E1 31807.732,E2 31807.732} C_VEL
LIN {X 0,Y 707.036,Z 853.64,A -85,B 0,C 180,E1 31807.075,E2 31807.075} C_VEL
LIN {X 0,Y 706.273,Z 876.461,A -85,B 0,C 180,E1 31806.384,E2 31806.384} C_VEL
LIN {X 0,Y 705.446,Z 900.25,A -85,B 0,C 180,E1 31805.53,E2 31805.53} C_VEL
LIN {X 0,Y 704.47,Z 925.785,A -85,B 0,C 180,E1 31804.447,E2 31804.447} C_VEL
LIN {X 0,Y 703.454,Z 949.024,A -85,B 0,C 180,E1 31803.302,E2 31803.302} C_VEL
LIN {X 0,Y 702.466,Z 971.076,A -85,B 0,C 180,E1 31802.069,E2 31802.069} C_VEL
LIN {X 0,Y 701.434,Z 994.98,A -85,B 0,C 180,E1 31800.544,E2 31800.544} C_VEL
LIN {X 0,Y 700.436,Z 1017.125,A -85,B 0,C 180,E1 31798.943,E2 31798.943} C_VEL
LIN {X 0,Y 699.469,Z 1039.286,A -85,B 0,C 180,E1 31797.131,E2 31797.131} C_VEL
LIN {X 0,Y 698.672,Z 1058.729,A -85,B 0,C 180,E1 31795.336,E2 31795.336} C_VEL
LIN {X 0,Y 697.94,Z 1078.324,A -85,B 0,C 180,E1 31793.292,E2 31793.292} C_VEL
LIN {X 0,Y 697.429,Z 1092.593,A -85,B 0,C 180,E1 31791.621,E2 31791.621} C_VEL
LIN {X 0,Y 697.038,Z 1105.392,A -85,B 0,C 180,E1 31789.963,E2 31789.963} C_VEL
LIN {X 0,Y 696.664,Z 1119.745,A -85,B 0,C 180,E1 31787.888,E2 31787.888} C_VEL
LIN {X 0,Y 696.376,Z 1131.944,A -85,B 0,C 180,E1 31785.832,E2 31785.832} C_VEL
LIN {X 0,Y 696.19,Z 1141.25,A -85,B 0,C 180,E1 31784.048,E2 31784.048} C_VEL
LIN {X 0,Y 696.081,Z 1148.953,A -85,B 0,C 180,E1 31782.36,E2 31782.36} C_VEL
LIN {X 0,Y 695.999,Z 1156.255,A -85,B 0,C 180,E1 31780.513,E2 31780.513} C_VEL
LIN {X 0,Y 695.957,Z 1163.207,A -85,B 0,C 180,E1 31778.344,E2 31778.344} C_VEL
LIN {X 0,Y 695.927,Z 1168.676,A -85,B 0,C 180,E1 31776.104,E2 31776.104} C_VEL
LIN {X 0,Y 695.913,Z 1172.312,A -85,B 0,C 180,E1 31773.956,E2 31773.956} C_VEL
LIN {X 0,Y 695.907,Z 1174.447,A -85,B 0,C 180,E1 31771.73,E2 31771.73} C_VEL
LIN {X 0,Y 695.89,Z 1174.907,A -85,B 0,C 180,E1 31769.507,E2 31769.507} C_VEL
LIN {X 0,Y 695.907,Z 1173.876,A -85,B 0,C 180,E1 31767.366,E2 31767.366} C_VEL
LIN {X 0,Y 695.917,Z 1170.989,A -85,B 0,C 180,E1 31765.056,E2 31765.056} C_VEL
LIN {X 0,Y 695.932,Z 1166.656,A -85,B 0,C 180,E1 31762.903,E2 31762.903} C_VEL
LIN {X 0,Y 695.963,Z 1161.024,A -85,B 0,C 180,E1 31760.825,E2 31760.825} C_VEL
LIN {X 0,Y 696.047,Z 1153.177,A -85,B 0,C 180,E1 31758.567,E2 31758.567} C_VEL
LIN {X 0,Y 696.16,Z 1143.338,A -85,B 0,C 180,E1 31756.292,E2 31756.292} C_VEL
LIN {X 0,Y 696.322,Z 1134.14,A -85,B 0,C 180,E1 31754.479,E2 31754.479} C_VEL
LIN {X 0,Y 696.532,Z 1124.485,A -85,B 0,C 180,E1 31752.801,E2 31752.801} C_VEL
LIN {X 0,Y 696.807,Z 1113.971,A -85,B 0,C 180,E1 31751.165,E2 31751.165} C_VEL
LIN {X 0,Y 697.143,Z 1101.557,A -85,B 0,C 180,E1 31749.429,E2 31749.429} C_VEL
LIN {X 0,Y 697.697,Z 1084.59,A -85,B 0,C 180,E1 31747.326,E2 31747.326} C_VEL
LIN {X 0,Y 698.301,Z 1068.43,A -85,B 0,C 180,E1 31745.557,E2 31745.557} C_VEL
LIN {X 0,Y 698.975,Z 1050.782,A -85,B 0,C 180,E1 31743.814,E2 31743.814} C_VEL
LIN {X 0,Y 699.882,Z 1030.013,A -85,B 0,C 180,E1 31741.996,E2 31741.996} C_VEL
LIN {X 0,Y 700.816,Z 1008.635,A -85,B 0,C 180,E1 31740.326,E2 31740.326} C_VEL
LIN {X 0,Y 701.836,Z 985.522,A -85,B 0,C 180,E1 31738.739,E2 31738.739} C_VEL
LIN {X 0,Y 702.822,Z 963.829,A -85,B 0,C 180,E1 31737.421,E2 31737.421} C_VEL
LIN {X 0,Y 703.88,Z 939.472,A -85,B 0,C 180,E1 31736.114,E2 31736.114} C_VEL
LIN {X 0,Y 704.86,Z 915.033,A -85,B 0,C 180,E1 31734.986,E2 31734.986} C_VEL
LIN {X 0,Y 705.726,Z 892.518,A -85,B 0,C 180,E1 31734.088,E2 31734.088} C_VEL
LIN {X 0,Y 706.661,Z 866.099,A -85,B 0,C 180,E1 31733.192,E2 31733.192} C_VEL
LIN {X 0,Y 707.443,Z 839.278,A -85,B 0,C 180,E1 31732.467,E2 31732.467} C_VEL
LIN {X 0,Y 708.033,Z 814.503,A -85,B 0,C 180,E1 31731.943,E2 31731.943} C_VEL
LIN {X 0,Y 708.513,Z 787.853,A -85,B 0,C 180,E1 31731.531,E2 31731.531} C_VEL
LIN {X 0,Y 710.397,Z 559.384,A -85,B 0,C 180,E1 31728.704,E2 31728.704} C_VEL
LIN {X 0,Y 712.222,Z 350.755,A -85,B 0,C 180,E1 31726.036,E2 31726.036} C_VEL
LIN {X 0,Y 712.142,Z 342.651,A -85,B 0,C 180,E1 31725.919,E2 31725.919} C_VEL
LIN {X 0,Y 700.557,Z 325.355,A -85,B 0,C 180,E1 31724.75,E2 31724.75} C_VEL
LIN {X 0,Y 697.437,Z 320.591,A -85,B 0,C 180,E1 31724.398,E2 31724.398} C_VEL
LIN {X 0,Y 696.389,Z 317.49,A -85,B 0,C 180,E1 31724.045,E2 31724.045} C_VEL
LIN {X 0,Y 696.375,Z 317.491,A -85,B 0,C 180,E1 31721.08,E2 31721.08} C_VEL
LIN {X 0,Y 696.384,Z 317.49,A -85,B 0,C 180,E1 31718.232,E2 31718.232} C_VEL
LIN {X 0,Y 696.391,Z 317.487,A -85,B 0,C 180,E1 31715.254,E2 31715.254} C_VEL
LIN {X 0,Y 696.398,Z 317.481,A -85,B 0,C 180,E1 31712.187,E2 31712.187} C_VEL
LIN {X 0,Y 696.399,Z 317.464,A -85,B 0,C 180,E1 31709.126,E2 31709.126} C_VEL
LIN {X 0,Y 696.394,Z 317.482,A -85,B 0,C 180,E1 31706.155,E2 31706.155} C_VEL
LIN {X 0,Y 696.407,Z 317.484,A -85,B 0,C 180,E1 31702.988,E2 31702.988} C_VEL
LIN {X 0,Y 696.376,Z 317.47,A -85,B 0,C 180,E1 31700.07,E2 31700.07} C_VEL
LIN {X 0,Y 696.4,Z 317.483,A -85,B 0,C 180,E1 31697.019,E2 31697.019} C_VEL
LIN {X 0,Y 696.372,Z 317.487,A -85,B 0,C 180,E1 31694.044,E2 31694.044} C_VEL
LIN {X 0,Y 696.398,Z 317.467,A -85,B 0,C 180,E1 31691.093,E2 31691.093} C_VEL
LIN {X 0,Y 696.372,Z 317.489,A -85,B 0,C 180,E1 31688.089,E2 31688.089} C_VEL
LIN {X 0,Y 696.4,Z 317.475,A -85,B 0,C 180,E1 31685.19,E2 31685.19} C_VEL
LIN {X 0,Y 696.386,Z 317.472,A -85,B 0,C 180,E1 31682.139,E2 31682.139} C_VEL
LIN {X 0,Y 696.396,Z 317.487,A -85,B 0,C 180,E1 31679.177,E2 31679.177} C_VEL
LIN {X 0,Y 696.402,Z 317.48,A -85,B 0,C 180,E1 31675.966,E2 31675.966} C_VEL
LIN {X 0,Y 696.373,Z 317.467,A -85,B 0,C 180,E1 31673.073,E2 31673.073} C_VEL
LIN {X 0,Y 696.402,Z 317.473,A -85,B 0,C 180,E1 31669.995,E2 31669.995} C_VEL
LIN {X 0,Y 696.372,Z 317.488,A -85,B 0,C 180,E1 31667.056,E2 31667.056} C_VEL
LIN {X 0,Y 696.402,Z 317.481,A -85,B 0,C 180,E1 31664.083,E2 31664.083} C_VEL
LIN {X 0,Y 696.382,Z 317.492,A -85,B 0,C 180,E1 31663.27,E2 31663.27} C_VEL
LIN {X 0,Y 697.733,Z 321.002,A -85,B 0,C 180,E1 31662.744,E2 31662.744} C_VEL
LIN {X 0,Y 699.189,Z 323.065,A -85,B 0,C 180,E1 31662.351,E2 31662.351} C_VEL
LIN {X 0,Y 701.247,Z 326.936,A -85,B 0,C 180,E1 31661.718,E2 31661.718} C_VEL
LIN {X 0,Y 703.897,Z 331.845,A -85,B 0,C 180,E1 31660.93,E2 31660.93} C_VEL
LIN {X 0,Y 709.797,Z 343.316,A -85,B 0,C 180,E1 31659.207,E2 31659.207} C_VEL
LIN {X 0,Y 713.063,Z 349.692,A -85,B 0,C 180,E1 31658.294,E2 31658.294} C_VEL
LIN {X 0,Y 711.656,Z 384.067,A -85,B 0,C 180,E1 31655.646,E2 31655.646} C_VEL
LIN {X 0,Y 710.274,Z 420.103,A -85,B 0,C 180,E1 31653.009,E2 31653.009} C_VEL
LIN {X 0,Y 708.914,Z 457.19,A -85,B 0,C 180,E1 31650.418,E2 31650.418} C_VEL
LIN {X 0,Y 707.617,Z 496.754,A -85,B 0,C 180,E1 31647.763,E2 31647.763} C_VEL
LIN {X 0,Y 706.725,Z 538.501,A -85,B 0,C 180,E1 31645.04,E2 31645.04} C_VEL
LIN {X 0,Y 708.172,Z 550.213,A -85,B 0,C 180,E1 31644.179,E2 31644.179} C_VEL
LIN {X 0,Y 711.031,Z 559.443,A -85,B 0,C 180,E1 31643.398,E2 31643.398} C_VEL
LIN {X 0,Y 715.25,Z 567.024,A -85,B 0,C 180,E1 31642.647,E2 31642.647} C_VEL
LIN {X 0,Y 721.029,Z 573.347,A -85,B 0,C 180,E1 31641.895,E2 31641.895} C_VEL
LIN {X 0,Y 726.984,Z 577.487,A -85,B 0,C 180,E1 31641.258,E2 31641.258} C_VEL
LIN {X 0,Y 730.272,Z 578.629,A -85,B 0,C 180,E1 31640.8,E2 31640.8} C_VEL
LIN {X 0,Y 732.553,Z 578.339,A -85,B 0,C 180,E1 31640.298,E2 31640.298} C_VEL
LIN {X 0,Y 733.512,Z 576.948,A -85,B 0,C 180,E1 31639.851,E2 31639.851} C_VEL
LIN {X 0,Y 733.398,Z 574.444,A -85,B 0,C 180,E1 31639.408,E2 31639.408} C_VEL
LIN {X 0,Y 731.982,Z 570.723,A -85,B 0,C 180,E1 31638.983,E2 31638.983} C_VEL
LIN {X 0,Y 729.277,Z 566.032,A -85,B 0,C 180,E1 31638.639,E2 31638.639} C_VEL
LIN {X 0,Y 723.58,Z 556.742,A -85,B 0,C 180,E1 31638.231,E2 31638.231} C_VEL
LIN {X 0,Y 718.839,Z 545.992,A -85,B 0,C 180,E1 31637.892,E2 31637.892} C_VEL
LIN {X 0,Y 715.23,Z 533.892,A -85,B 0,C 180,E1 31637.63,E2 31637.63} C_VEL
LIN {X 0,Y 712.832,Z 520.333,A -85,B 0,C 180,E1 31637.454,E2 31637.454} C_VEL
LIN {X 0,Y 711.676,Z 504.838,A -85,B 0,C 180,E1 31637.369,E2 31637.369} C_VEL
LIN {X 0,Y 711.544,Z 338.132,A -85,B 0,C 180,E1 31637.359,E2 31637.359} C_VEL
LIN {X 0,Y 705.681,Z 331.015,A -85,B 0,C 180,E1 31636.919,E2 31636.919} C_VEL
LIN {X 0,Y 702.947,Z 330.603,A -85,B 0,C 180,E1 31636.71,E2 31636.71} C_VEL
LIN {X 0,Y 702.218,Z 330.122,A -85,B 0,C 180,E1 31636.646,E2 31636.646} C_VEL
LIN {X 0,Y 708.138,Z 343.433,A -85,B 0,C 180,E1 31635.172,E2 31635.172} C_VEL
LIN {X 0,Y 708.015,Z 351.108,A -85,B 0,C 180,E1 31634.66,E2 31634.66} C_VEL
LIN {X 0,Y 712.348,Z 368.549,A -85,B 0,C 180,E1 31634.076,E2 31634.076} C_VEL
LIN {X 0,Y 710.479,Z 579.097,A -85,B 0,C 180,E1 31631.381,E2 31631.381} C_VEL
LIN {X 0,Y 708.655,Z 802.749,A -85,B 0,C 180,E1 31628.61,E2 31628.61} C_VEL
LIN {X 0,Y 708.238,Z 835.904,A -85,B 0,C 180,E1 31628.164,E2 31628.164} C_VEL
LIN {X 0,Y 707.6,Z 863.323,A -85,B 0,C 180,E1 31627.629,E2 31627.629} C_VEL
LIN {X 0,Y 706.868,Z 889.39,A -85,B 0,C 180,E1 31626.959,E2 31626.959} C_VEL
LIN {X 0,Y 705.977,Z 916.985,A -85,B 0,C 180,E1 31626.07,E2 31626.07} C_VEL
LIN {X 0,Y 705.061,Z 940.694,A -85,B 0,C 180,E1 31625.152,E2 31625.152} C_VEL
LIN {X 0,Y 704.142,Z 962.734,A -85,B 0,C 180,E1 31624.166,E2 31624.166} C_VEL
LIN {X 0,Y 703.1,Z 987.357,A -85,B 0,C 180,E1 31622.903,E2 31622.903} C_VEL
LIN {X 0,Y 702.088,Z 1010.099,A -85,B 0,C 180,E1 31621.558,E2 31621.558} C_VEL
LIN {X 0,Y 701.211,Z 1029.613,A -85,B 0,C 180,E1 31620.268,E2 31620.268} C_VEL
LIN {X 0,Y 700.237,Z 1051.264,A -85,B 0,C 180,E1 31618.67,E2 31618.67} C_VEL
LIN {X 0,Y 699.358,Z 1072.248,A -85,B 0,C 180,E1 31616.912,E2 31616.912} C_VEL
LIN {X 0,Y 698.605,Z 1090.226,A -85,B 0,C 180,E1 31615.235,E2 31615.235} C_VEL
LIN {X 0,Y 697.92,Z 1108.725,A -85,B 0,C 180,E1 31613.29,E2 31613.29} C_VEL
LIN {X 0,Y 697.413,Z 1122.98,A -85,B 0,C 180,E1 31611.619,E2 31611.619} C_VEL
LIN {X 0,Y 696.979,Z 1137.697,A -85,B 0,C 180,E1 31609.701,E2 31609.701} C_VEL
LIN {X 0,Y 696.597,Z 1152.15,A -85,B 0,C 180,E1 31607.542,E2 31607.542} C_VEL
LIN {X 0,Y 696.353,Z 1163.148,A -85,B 0,C 180,E1 31605.66,E2 31605.66} C_VEL
LIN {X 0,Y 696.173,Z 1172.732,A -85,B 0,C 180,E1 31603.792,E2 31603.792} C_VEL
LIN {X 0,Y 696.046,Z 1182.006,A -85,B 0,C 180,E1 31601.685,E2 31601.685} C_VEL
LIN {X 0,Y 695.972,Z 1189.82,A -85,B 0,C 180,E1 31599.509,E2 31599.509} C_VEL
LIN {X 0,Y 695.937,Z 1195.973,A -85,B 0,C 180,E1 31597.345,E2 31597.345} C_VEL
LIN {X 0,Y 695.922,Z 1200.64,A -85,B 0,C 180,E1 31595.11,E2 31595.11} C_VEL
LIN {X 0,Y 695.918,Z 1203.516,A -85,B 0,C 180,E1 31592.964,E2 31592.964} C_VEL
LIN {X 0,Y 695.906,Z 1204.775,A -85,B 0,C 180,E1 31590.905,E2 31590.905} C_VEL
LIN {X 0,Y 695.906,Z 1204.775,A -85,B 0,C 180,E1 31589.093,E2 31589.093} C_VEL
LIN {X 0,Y 695.918,Z 1203.514,A -85,B 0,C 180,E1 31587.034,E2 31587.034} C_VEL
LIN {X 0,Y 695.923,Z 1200.636,A -85,B 0,C 180,E1 31584.888,E2 31584.888} C_VEL
LIN {X 0,Y 695.936,Z 1195.969,A -85,B 0,C 180,E1 31582.652,E2 31582.652} C_VEL
LIN {X 0,Y 695.973,Z 1189.813,A -85,B 0,C 180,E1 31580.489,E2 31580.489} C_VEL
LIN {X 0,Y 696.046,Z 1181.998,A -85,B 0,C 180,E1 31578.313,E2 31578.313} C_VEL
LIN {X 0,Y 696.174,Z 1172.722,A -85,B 0,C 180,E1 31576.206,E2 31576.206} C_VEL
LIN {X 0,Y 696.353,Z 1163.136,A -85,B 0,C 180,E1 31574.338,E2 31574.338} C_VEL
LIN {X 0,Y 696.614,Z 1151.614,A -85,B 0,C 180,E1 31572.37,E2 31572.37} C_VEL
LIN {X 0,Y 697,Z 1137.036,A -85,B 0,C 180,E1 31570.21,E2 31570.21} C_VEL
LIN {X 0,Y 697.412,Z 1122.963,A -85,B 0,C 180,E1 31568.378,E2 31568.378} C_VEL
LIN {X 0,Y 697.952,Z 1107.926,A -85,B 0,C 180,E1 31566.619,E2 31566.619} C_VEL
LIN {X 0,Y 698.693,Z 1088.255,A -85,B 0,C 180,E1 31564.575,E2 31564.575} C_VEL
LIN {X 0,Y 699.432,Z 1070.285,A -85,B 0,C 180,E1 31562.914,E2 31562.914} C_VEL
LIN {X 0,Y 700.395,Z 1048.251,A -85,B 0,C 180,E1 31561.097,E2 31561.097} C_VEL
LIN {X 0,Y 701.338,Z 1026.931,A -85,B 0,C 180,E1 31559.546,E2 31559.546} C_VEL
LIN {X 0,Y 702.35,Z 1004.19,A -85,B 0,C 180,E1 31558.069,E2 31558.069} C_VEL
LIN {X 0,Y 703.417,Z 979.988,A -85,B 0,C 180,E1 31556.703,E2 31556.703} C_VEL
LIN {X 0,Y 704.329,Z 958.709,A -85,B 0,C 180,E1 31555.645,E2 31555.645} C_VEL
LIN {X 0,Y 705.327,Z 934.762,A -85,B 0,C 180,E1 31554.601,E2 31554.601} C_VEL
LIN {X 0,Y 706.244,Z 907.801,A -85,B 0,C 180,E1 31553.614,E2 31553.614} C_VEL
LIN {X 0,Y 707.072,Z 883.048,A -85,B 0,C 180,E1 31552.861,E2 31552.861} C_VEL
LIN {X 0,Y 707.784,Z 856.194,A -85,B 0,C 180,E1 31552.216,E2 31552.216} C_VEL
LIN {X 0,Y 708.329,Z 829.428,A -85,B 0,C 180,E1 31551.736,E2 31551.736} C_VEL
LIN {X 0,Y 709.93,Z 643.969,A -85,B 0,C 180,E1 31549.432,E2 31549.432} C_VEL
LIN {X 0,Y 711.708,Z 435.819,A -85,B 0,C 180,E1 31546.793,E2 31546.793} C_VEL
LIN {X 0,Y 712.364,Z 349.877,A -85,B 0,C 180,E1 31545.668,E2 31545.668} C_VEL
LIN {X 0,Y 712.168,Z 342.01,A -85,B 0,C 180,E1 31545.515,E2 31545.515} C_VEL
LIN {X 0,Y 702.209,Z 327.252,A -85,B 0,C 180,E1 31544.387,E2 31544.387} C_VEL
LIN {X 0,Y 699.716,Z 323.121,A -85,B 0,C 180,E1 31544.087,E2 31544.087} C_VEL
LIN {X 0,Y 697.135,Z 320.027,A -85,B 0,C 180,E1 31543.798,E2 31543.798} C_VEL
LIN {X 0,Y 696.938,Z 319.601,A -85,B 0,C 180,E1 31543.757,E2 31543.757} C_VEL
LIN {X 0,Y 698.965,Z 322.459,A -85,B 0,C 180,E1 31543.594,E2 31543.594} C_VEL
LIN {X 0,Y 701.598,Z 324.031,A -85,B 0,C 180,E1 31543.319,E2 31543.319} C_VEL
LIN {X 0,Y 703.976,Z 327.234,A -85,B 0,C 180,E1 31542.899,E2 31542.899} C_VEL
LIN {X 0,Y 705.176,Z 328.681,A -85,B 0,C 180,E1 31542.449,E2 31542.449} C_VEL
LIN {X 0,Y 705.265,Z 328.929,A -85,B 0,C 180,E1 31542.004,E2 31542.004} C_VEL
LIN {X 0,Y 704.248,Z 328.118,A -85,B 0,C 180,E1 31541.533,E2 31541.533} C_VEL
LIN {X 0,Y 702.327,Z 325.951,A -85,B 0,C 180,E1 31541.101,E2 31541.101} C_VEL
LIN {X 0,Y 700.544,Z 323.528,A -85,B 0,C 180,E1 31540.822,E2 31540.822} C_VEL
LIN {X 0,Y 697.875,Z 321.187,A -85,B 0,C 180,E1 31540.524,E2 31540.524} C_VEL
LIN {X 0,Y 696.474,Z 317.919,A -85,B 0,C 180,E1 31540.323,E2 31540.323} C_VEL
LIN {X 0,Y 696.403,Z 317.466,A -85,B 0,C 180,E1 31540.271,E2 31540.271} C_VEL
LIN {X 0,Y 696.384,Z 317.465,A -85,B 0,C 180,E1 31537.399,E2 31537.399} C_VEL
LIN {X 0,Y 696.401,Z 317.486,A -85,B 0,C 180,E1 31534.252,E2 31534.252} C_VEL
LIN {X 0,Y 696.4,Z 317.458,A -85,B 0,C 180,E1 31531.159,E2 31531.159} C_VEL
LIN {X 0,Y 696.396,Z 317.487,A -85,B 0,C 180,E1 31528.096,E2 31528.096} C_VEL
LIN {X 0,Y 696.368,Z 317.457,A -85,B 0,C 180,E1 31525.152,E2 31525.152} C_VEL
LIN {X 0,Y 696.406,Z 317.489,A -85,B 0,C 180,E1 31522.167,E2 31522.167} C_VEL
LIN {X 0,Y 696.37,Z 317.489,A -85,B 0,C 180,E1 31519.197,E2 31519.197} C_VEL
LIN {X 0,Y 696.379,Z 317.484,A -85,B 0,C 180,E1 31516.345,E2 31516.345} C_VEL
LIN {X 0,Y 696.402,Z 317.488,A -85,B 0,C 180,E1 31513.281,E2 31513.281} C_VEL
LIN {X 0,Y 696.409,Z 317.63,A -85,B 0,C 180,E1 31511.659,E2 31511.659} C_VEL
LIN {X 0,Y 697.74,Z 323.96,A -85,B 0,C 180,E1 31511.42,E2 31511.42} C_VEL
LIN {X 0,Y 697.792,Z 399.797,A -85,B 0,C 180,E1 31508.82,E2 31508.82} C_VEL
LIN {X 0,Y 698.207,Z 484.241,A -85,B 0,C 180,E1 31505.795,E2 31505.795} C_VEL
LIN {X 0,Y 698.432,Z 555.496,A -85,B 0,C 180,E1 31503.16,E2 31503.16} C_VEL
LIN {X 0,Y 698.235,Z 634.755,A -85,B 0,C 180,E1 31500.164,E2 31500.164} C_VEL
LIN {X 0,Y 697.795,Z 711.826,A -85,B 0,C 180,E1 31497.207,E2 31497.207} C_VEL
LIN {X 0,Y 697.266,Z 789.709,A -85,B 0,C 180,E1 31494.198,E2 31494.198} C_VEL
LIN {X 0,Y 696.953,Z 837.537,A -85,B 0,C 180,E1 31492.349,E2 31492.349} C_VEL
LIN {X 0,Y 696.848,Z 942.817,A -85,B 0,C 180,E1 31491.27,E2 31491.27} C_VEL
LIN {X 0,Y 695.847,Z 950.471,A -85,B 0,C 180,E1 31491.193,E2 31491.193} C_VEL
LIN {X 0,Y 691.037,Z 965.172,A -85,B 0,C 180,E1 31490.99,E2 31490.99} C_VEL
LIN {X 0,Y 689.013,Z 973.524,A -85,B 0,C 180,E1 31490.794,E2 31490.794} C_VEL
LIN {X 0,Y 688.789,Z 976.609,A -85,B 0,C 180,E1 31490.7,E2 31490.7} C_VEL
LIN {X 0,Y 688.667,Z 989.058,A -85,B 0,C 180,E1 31490.219,E2 31490.219} C_VEL
LIN {X 0,Y 688.5,Z 1001.61,A -85,B 0,C 180,E1 31489.583,E2 31489.583} C_VEL
LIN {X 0,Y 688.355,Z 1014.376,A -85,B 0,C 180,E1 31488.733,E2 31488.733} C_VEL
LIN {X 0,Y 688.215,Z 1024.107,A -85,B 0,C 180,E1 31487.901,E2 31487.901} C_VEL
LIN {X 0,Y 688.095,Z 1033.478,A -85,B 0,C 180,E1 31486.898,E2 31486.898} C_VEL
LIN {X 0,Y 688.006,Z 1040.781,A -85,B 0,C 180,E1 31485.868,E2 31485.868} C_VEL
LIN {X 0,Y 687.963,Z 1045.993,A -85,B 0,C 180,E1 31484.92,E2 31484.92} C_VEL
LIN {X 0,Y 687.937,Z 1050.277,A -85,B 0,C 180,E1 31483.882,E2 31483.882} C_VEL
LIN {X 0,Y 687.915,Z 1053.724,A -85,B 0,C 180,E1 31482.577,E2 31482.577} C_VEL
LIN {X 0,Y 687.917,Z 1054.987,A -85,B 0,C 180,E1 31481.527,E2 31481.527} C_VEL
LIN {X 0,Y 687.916,Z 1055.028,A -85,B 0,C 180,E1 31480.47,E2 31480.47} C_VEL
LIN {X 0,Y 687.915,Z 1053.687,A -85,B 0,C 180,E1 31479.317,E2 31479.317} C_VEL
LIN {X 0,Y 687.938,Z 1050.218,A -85,B 0,C 180,E1 31478.019,E2 31478.019} C_VEL
LIN {X 0,Y 687.962,Z 1045.934,A -85,B 0,C 180,E1 31476.985,E2 31476.985} C_VEL
LIN {X 0,Y 688.007,Z 1040.401,A -85,B 0,C 180,E1 31475.988,E2 31475.988} C_VEL
LIN {X 0,Y 688.104,Z 1032.107,A -85,B 0,C 180,E1 31474.862,E2 31474.862} C_VEL
LIN {X 0,Y 688.215,Z 1023.383,A -85,B 0,C 180,E1 31473.95,E2 31473.95} C_VEL
LIN {X 0,Y 688.354,Z 1013.426,A -85,B 0,C 180,E1 31473.111,E2 31473.111} C_VEL
LIN {X 0,Y 688.501,Z 1001.133,A -85,B 0,C 180,E1 31472.307,E2 31472.307} C_VEL
LIN {X 0,Y 688.657,Z 989.076,A -85,B 0,C 180,E1 31471.698,E2 31471.698} C_VEL
LIN {X 0,Y 688.79,Z 975.808,A -85,B 0,C 180,E1 31471.187,E2 31471.187} C_VEL
LIN {X 0,Y 688.899,Z 961.093,A -85,B 0,C 180,E1 31470.799,E2 31470.799} C_VEL
LIN {X 0,Y 688.958,Z 946.012,A -85,B 0,C 180,E1 31470.559,E2 31470.559} C_VEL
LIN {X 0,Y 689.081,Z 837.454,A -85,B 0,C 180,E1 31469.43,E2 31469.43} C_VEL
LIN {X 0,Y 689.73,Z 757.012,A -85,B 0,C 180,E1 31466.273,E2 31466.273} C_VEL
LIN {X 0,Y 690.309,Z 677.23,A -85,B 0,C 180,E1 31463.18,E2 31463.18} C_VEL
LIN {X 0,Y 690.904,Z 600.794,A -85,B 0,C 180,E1 31460.179,E2 31460.179} C_VEL
LIN {X 0,Y 691.392,Z 523.719,A -85,B 0,C 180,E1 31457.158,E2 31457.158} C_VEL
LIN {X 0,Y 691.548,Z 448.008,A -85,B 0,C 180,E1 31454.209,E2 31454.209} C_VEL
LIN {X 0,Y 691.588,Z 447.023,A -85,B 0,C 180,E1 31454.161,E2 31454.161} C_VEL
LIN {X 0,Y 692.733,Z 448.849,A -85,B 0,C 180,E1 31454.043,E2 31454.043} C_VEL
LIN {X 0,Y 694.511,Z 449.08,A -85,B 0,C 180,E1 31453.898,E2 31453.898} C_VEL
LIN {X 0,Y 697.202,Z 447.105,A -85,B 0,C 180,E1 31453.713,E2 31453.713} C_VEL
LIN {X 0,Y 700.713,Z 441.958,A -85,B 0,C 180,E1 31453.51,E2 31453.51} C_VEL
LIN {X 0,Y 701.323,Z 441.167,A -85,B 0,C 180,E1 31453.473,E2 31453.473} C_VEL
LIN {X 0,Y 704.876,Z 439.961,A -85,B 0,C 180,E1 31453.216,E2 31453.216} C_VEL
LIN {X 0,Y 705.525,Z 439.716,A -85,B 0,C 180,E1 31453.17,E2 31453.17} C_VEL
LIN {X 0,Y 703.536,Z 647.449,A -85,B 0,C 180,E1 31450.528,E2 31450.528} C_VEL
LIN {X 0,Y 702.037,Z 799.329,A -85,B 0,C 180,E1 31448.626,E2 31448.626} C_VEL
LIN {X 0,Y 701.425,Z 826.602,A -85,B 0,C 180,E1 31448.135,E2 31448.135} C_VEL
LIN {X 0,Y 700.583,Z 853.588,A -85,B 0,C 180,E1 31447.476,E2 31447.476} C_VEL
LIN {X 0,Y 699.73,Z 876.473,A -85,B 0,C 180,E1 31446.78,E2 31446.78} C_VEL
LIN {X 0,Y 698.766,Z 900.51,A -85,B 0,C 180,E1 31445.912,E2 31445.912} C_VEL
LIN {X 0,Y 697.625,Z 926.835,A -85,B 0,C 180,E1 31444.782,E2 31444.782} C_VEL
LIN {X 0,Y 696.518,Z 949.522,A -85,B 0,C 180,E1 31443.651,E2 31443.651} C_VEL
LIN {X 0,Y 695.431,Z 971.079,A -85,B 0,C 180,E1 31442.433,E2 31442.433} C_VEL
LIN {X 0,Y 694.201,Z 995.547,A -85,B 0,C 180,E1 31440.857,E2 31440.857} C_VEL
LIN {X 0,Y 693.109,Z 1017.139,A -85,B 0,C 180,E1 31439.279,E2 31439.279} C_VEL
LIN {X 0,Y 691.965,Z 1039.805,A -85,B 0,C 180,E1 31437.403,E2 31437.403} C_VEL
LIN {X 0,Y 691.061,Z 1059.671,A -85,B 0,C 180,E1 31435.543,E2 31435.543} C_VEL
LIN {X 0,Y 690.242,Z 1078.33,A -85,B 0,C 180,E1 31433.567,E2 31433.567} C_VEL
LIN {X 0,Y 689.667,Z 1092.599,A -85,B 0,C 180,E1 31431.877,E2 31431.877} C_VEL
LIN {X 0,Y 689.215,Z 1105.586,A -85,B 0,C 180,E1 31430.174,E2 31430.174} C_VEL
LIN {X 0,Y 688.762,Z 1120.159,A -85,B 0,C 180,E1 31428.032,E2 31428.032} C_VEL
LIN {X 0,Y 688.437,Z 1132.319,A -85,B 0,C 180,E1 31425.951,E2 31425.951} C_VEL
LIN {X 0,Y 688.248,Z 1141.253,A -85,B 0,C 180,E1 31424.214,E2 31424.214} C_VEL
LIN {X 0,Y 688.113,Z 1149.184,A -85,B 0,C 180,E1 31422.451,E2 31422.451} C_VEL
LIN {X 0,Y 688.009,Z 1156.552,A -85,B 0,C 180,E1 31420.552,E2 31420.552} C_VEL
LIN {X 0,Y 687.962,Z 1163.45,A -85,B 0,C 180,E1 31418.358,E2 31418.358} C_VEL
LIN {X 0,Y 687.926,Z 1169.021,A -85,B 0,C 180,E1 31416.008,E2 31416.008} C_VEL
LIN {X 0,Y 687.911,Z 1172.515,A -85,B 0,C 180,E1 31413.835,E2 31413.835} C_VEL
LIN {X 0,Y 687.907,Z 1174.493,A -85,B 0,C 180,E1 31411.667,E2 31411.667} C_VEL
LIN {X 0,Y 687.891,Z 1174.887,A -85,B 0,C 180,E1 31409.418,E2 31409.418} C_VEL
LIN {X 0,Y 687.908,Z 1173.876,A -85,B 0,C 180,E1 31407.335,E2 31407.335} C_VEL
LIN {X 0,Y 687.919,Z 1170.985,A -85,B 0,C 180,E1 31404.998,E2 31404.998} C_VEL
LIN {X 0,Y 687.933,Z 1166.848,A -85,B 0,C 180,E1 31402.904,E2 31402.904} C_VEL
LIN {X 0,Y 687.97,Z 1161.267,A -85,B 0,C 180,E1 31400.802,E2 31400.802} C_VEL
LIN {X 0,Y 688.057,Z 1153.813,A -85,B 0,C 180,E1 31398.602,E2 31398.602} C_VEL
LIN {X 0,Y 688.193,Z 1143.744,A -85,B 0,C 180,E1 31396.216,E2 31396.216} C_VEL
LIN {X 0,Y 688.394,Z 1134.305,A -85,B 0,C 180,E1 31394.327,E2 31394.327} C_VEL
LIN {X 0,Y 688.614,Z 1125.004,A -85,B 0,C 180,E1 31392.684,E2 31392.684} C_VEL
LIN {X 0,Y 688.93,Z 1114.55,A -85,B 0,C 180,E1 31391.029,E2 31391.029} C_VEL
LIN {X 0,Y 689.297,Z 1102.626,A -85,B 0,C 180,E1 31389.332,E2 31389.332} C_VEL
LIN {X 0,Y 689.863,Z 1087.582,A -85,B 0,C 180,E1 31387.41,E2 31387.41} C_VEL
LIN {X 0,Y 690.629,Z 1069.281,A -85,B 0,C 180,E1 31385.358,E2 31385.358} C_VEL
LIN {X 0,Y 691.391,Z 1051.73,A -85,B 0,C 180,E1 31383.597,E2 31383.597} C_VEL
LIN {X 0,Y 692.437,Z 1030.757,A -85,B 0,C 180,E1 31381.731,E2 31381.731} C_VEL
LIN {X 0,Y 693.53,Z 1008.622,A -85,B 0,C 180,E1 31379.983,E2 31379.983} C_VEL
LIN {X 0,Y 694.73,Z 985.18,A -85,B 0,C 180,E1 31378.36,E2 31378.36} C_VEL
LIN {X 0,Y 695.857,Z 963.022,A -85,B 0,C 180,E1 31377.005,E2 31377.005} C_VEL
LIN {X 0,Y 697.08,Z 937.513,A -85,B 0,C 180,E1 31375.639,E2 31375.639} C_VEL
LIN {X 0,Y 698.164,Z 914.553,A -85,B 0,C 180,E1 31374.578,E2 31374.578} C_VEL
LIN {X 0,Y 699.116,Z 892.507,A -85,B 0,C 180,E1 31373.695,E2 31373.695} C_VEL
LIN {X 0,Y 700.13,Z 866.672,A -85,B 0,C 180,E1 31372.812,E2 31372.812} C_VEL
LIN {X 0,Y 701.018,Z 839.92,A -85,B 0,C 180,E1 31372.08,E2 31372.08} C_VEL
LIN {X 0,Y 701.68,Z 815.245,A -85,B 0,C 180,E1 31371.552,E2 31371.552} C_VEL
LIN {X 0,Y 702.214,Z 789.524,A -85,B 0,C 180,E1 31371.146,E2 31371.146} C_VEL
LIN {X 0,Y 704.36,Z 560.846,A -85,B 0,C 180,E1 31368.291,E2 31368.291} C_VEL
LIN {X 0,Y 706.438,Z 351.979,A -85,B 0,C 180,E1 31365.6,E2 31365.6} C_VEL
LIN {X 0,Y 706.362,Z 346.35,A -85,B 0,C 180,E1 31365.516,E2 31365.516} C_VEL
LIN {X 0,Y 695.716,Z 330.501,A -85,B 0,C 180,E1 31364.421,E2 31364.421} C_VEL
LIN {X 0,Y 689.057,Z 320.656,A -85,B 0,C 180,E1 31363.688,E2 31363.688} C_VEL
LIN {X 0,Y 688.449,Z 318.479,A -85,B 0,C 180,E1 31363.434,E2 31363.434} C_VEL
LIN {X 0,Y 688.465,Z 318.478,A -85,B 0,C 180,E1 31360.372,E2 31360.372} C_VEL
LIN {X 0,Y 688.46,Z 318.476,A -85,B 0,C 180,E1 31357.263,E2 31357.263} C_VEL
LIN {X 0,Y 688.45,Z 318.462,A -85,B 0,C 180,E1 31354.272,E2 31354.272} C_VEL
LIN {X 0,Y 688.468,Z 318.477,A -85,B 0,C 180,E1 31351.134,E2 31351.134} C_VEL
LIN {X 0,Y 688.434,Z 318.468,A -85,B 0,C 180,E1 31348.166,E2 31348.166} C_VEL
LIN {X 0,Y 688.461,Z 318.455,A -85,B 0,C 180,E1 31345.185,E2 31345.185} C_VEL
LIN {X 0,Y 688.433,Z 318.479,A -85,B 0,C 180,E1 31342.187,E2 31342.187} C_VEL
LIN {X 0,Y 688.468,Z 318.463,A -85,B 0,C 180,E1 31339.161,E2 31339.161} C_VEL
LIN {X 0,Y 688.442,Z 318.459,A -85,B 0,C 180,E1 31336.019,E2 31336.019} C_VEL
LIN {X 0,Y 688.465,Z 318.475,A -85,B 0,C 180,E1 31333.095,E2 31333.095} C_VEL
LIN {X 0,Y 688.459,Z 318.461,A -85,B 0,C 180,E1 31329.953,E2 31329.953} C_VEL
LIN {X 0,Y 688.458,Z 318.459,A -85,B 0,C 180,E1 31326.84,E2 31326.84} C_VEL
LIN {X 0,Y 688.449,Z 318.478,A -85,B 0,C 180,E1 31323.831,E2 31323.831} C_VEL
LIN {X 0,Y 688.44,Z 318.463,A -85,B 0,C 180,E1 31320.832,E2 31320.832} C_VEL
LIN {X 0,Y 688.444,Z 318.461,A -85,B 0,C 180,E1 31317.919,E2 31317.919} C_VEL
LIN {X 0,Y 688.439,Z 318.479,A -85,B 0,C 180,E1 31315.001,E2 31315.001} C_VEL
LIN {X 0,Y 688.446,Z 318.463,A -85,B 0,C 180,E1 31312.069,E2 31312.069} C_VEL
LIN {X 0,Y 688.437,Z 318.451,A -85,B 0,C 180,E1 31309.116,E2 31309.116} C_VEL
LIN {X 0,Y 688.465,Z 318.452,A -85,B 0,C 180,E1 31306.135,E2 31306.135} C_VEL
LIN {X 0,Y 688.461,Z 318.551,A -85,B 0,C 180,E1 31304.284,E2 31304.284} C_VEL
LIN {X 0,Y 689.751,Z 321.963,A -85,B 0,C 180,E1 31303.753,E2 31303.753} C_VEL
LIN {X 0,Y 691.228,Z 323.854,A -85,B 0,C 180,E1 31303.356,E2 31303.356} C_VEL
LIN {X 0,Y 693.148,Z 327.728,A -85,B 0,C 180,E1 31302.713,E2 31302.713} C_VEL
LIN {X 0,Y 694.187,Z 329.589,A -85,B 0,C 180,E1 31302.393,E2 31302.393} C_VEL
LIN {X 0,Y 696.998,Z 334.965,A -85,B 0,C 180,E1 31301.516,E2 31301.516} C_VEL
LIN {X 0,Y 699.661,Z 339.913,A -85,B 0,C 180,E1 31300.724,E2 31300.724} C_VEL
LIN {X 0,Y 704.02,Z 348.13,A -85,B 0,C 180,E1 31299.463,E2 31299.463} C_VEL
LIN {X 0,Y 707.234,Z 354.763,A -85,B 0,C 180,E1 31298.52,E2 31298.52} C_VEL
LIN {X 0,Y 705.632,Z 389.544,A -85,B 0,C 180,E1 31295.825,E2 31295.825} C_VEL
LIN {X 0,Y 704.086,Z 425.226,A -85,B 0,C 180,E1 31293.199,E2 31293.199} C_VEL
LIN {X 0,Y 702.516,Z 463.674,A -85,B 0,C 180,E1 31290.497,E2 31290.497} C_VEL
LIN {X 0,Y 700.997,Z 504.293,A -85,B 0,C 180,E1 31287.759,E2 31287.759} C_VEL
LIN {X 0,Y 700.1,Z 541.464,A -85,B 0,C 180,E1 31285.314,E2 31285.314} C_VEL
LIN {X 0,Y 701.457,Z 553.33,A -85,B 0,C 180,E1 31284.438,E2 31284.438} C_VEL
LIN {X 0,Y 704.357,Z 563.249,A -85,B 0,C 180,E1 31283.598,E2 31283.598} C_VEL
LIN {X 0,Y 708.409,Z 571.028,A -85,B 0,C 180,E1 31282.835,E2 31282.835} C_VEL
LIN {X 0,Y 713.972,Z 577.725,A -85,B 0,C 180,E1 31282.062,E2 31282.062} C_VEL
LIN {X 0,Y 721.094,Z 583.181,A -85,B 0,C 180,E1 31281.29,E2 31281.29} C_VEL
LIN {X 0,Y 724.668,Z 584.942,A -85,B 0,C 180,E1 31280.908,E2 31280.908} C_VEL
LIN {X 0,Y 727.51,Z 585.562,A -85,B 0,C 180,E1 31280.48,E2 31280.48} C_VEL
LIN {X 0,Y 729.533,Z 584.951,A -85,B 0,C 180,E1 31279.998,E2 31279.998} C_VEL
LIN {X 0,Y 730.335,Z 583.275,A -85,B 0,C 180,E1 31279.538,E2 31279.538} C_VEL
LIN {X 0,Y 729.907,Z 580.311,A -85,B 0,C 180,E1 31279.066,E2 31279.066} C_VEL
LIN {X 0,Y 728.095,Z 576.342,A -85,B 0,C 180,E1 31278.652,E2 31278.652} C_VEL
LIN {X 0,Y 725.071,Z 571.646,A -85,B 0,C 180,E1 31278.336,E2 31278.336} C_VEL
LIN {X 0,Y 718.931,Z 561.76,A -85,B 0,C 180,E1 31277.899,E2 31277.899} C_VEL
LIN {X 0,Y 713.892,Z 550.516,A -85,B 0,C 180,E1 31277.532,E2 31277.532} C_VEL
LIN {X 0,Y 709.982,Z 537.838,A -85,B 0,C 180,E1 31277.243,E2 31277.243} C_VEL
LIN {X 0,Y 707.348,Z 524.029,A -85,B 0,C 180,E1 31277.045,E2 31277.045} C_VEL
LIN {X 0,Y 705.943,Z 508.512,A -85,B 0,C 180,E1 31276.939,E2 31276.939} C_VEL
LIN {X 0,Y 705.718,Z 484.496,A -85,B 0,C 180,E1 31276.922,E2 31276.922} C_VEL
LIN {X 0,Y 705.589,Z 341.703,A -85,B 0,C 180,E1 31276.912,E2 31276.912} C_VEL
LIN {X 0,Y 703.493,Z 339.115,A -85,B 0,C 180,E1 31276.752,E2 31276.752} C_VEL
LIN {X 0,Y 700.948,Z 340.122,A -85,B 0,C 180,E1 31276.556,E2 31276.556} C_VEL
LIN {X 0,Y 698.411,Z 339.432,A -85,B 0,C 180,E1 31276.359,E2 31276.359} C_VEL
LIN {X 0,Y 698.079,Z 339.235,A -85,B 0,C 180,E1 31276.321,E2 31276.321} C_VEL
LIN {X 0,Y 701.713,Z 347.379,A -85,B 0,C 180,E1 31275.412,E2 31275.412} C_VEL
LIN {X 0,Y 701.706,Z 351.113,A -85,B 0,C 180,E1 31275.171,E2 31275.171} C_VEL
LIN {X 0,Y 706.568,Z 370.741,A -85,B 0,C 180,E1 31274.501,E2 31274.501} C_VEL
LIN {X 0,Y 704.453,Z 580.651,A -85,B 0,C 180,E1 31271.793,E2 31271.793} C_VEL
LIN {X 0,Y 702.389,Z 803.727,A -85,B 0,C 180,E1 31269.006,E2 31269.006} C_VEL
LIN {X 0,Y 701.921,Z 836.183,A -85,B 0,C 180,E1 31268.565,E2 31268.565} C_VEL
LIN {X 0,Y 701.211,Z 863.594,A -85,B 0,C 180,E1 31268.027,E2 31268.027} C_VEL
LIN {X 0,Y 700.38,Z 889.592,A -85,B 0,C 180,E1 31267.353,E2 31267.353} C_VEL
LIN {X 0,Y 699.357,Z 917.577,A -85,B 0,C 180,E1 31266.443,E2 31266.443} C_VEL
LIN {X 0,Y 698.359,Z 940.703,A -85,B 0,C 180,E1 31265.54,E2 31265.54} C_VEL
LIN {X 0,Y 697.375,Z 961.746,A -85,B 0,C 180,E1 31264.594,E2 31264.594} C_VEL
LIN {X 0,Y 696.204,Z 985.656,A -85,B 0,C 180,E1 31263.37,E2 31263.37} C_VEL
LIN {X 0,Y 695.014,Z 1009.374,A -85,B 0,C 180,E1 31261.965,E2 31261.965} C_VEL
LIN {X 0,Y 693.995,Z 1029.618,A -85,B 0,C 180,E1 31260.616,E2 31260.616} C_VEL
LIN {X 0,Y 692.897,Z 1051.26,A -85,B 0,C 180,E1 31259.002,E2 31259.002} C_VEL
LIN {X 0,Y 691.859,Z 1072.345,A -85,B 0,C 180,E1 31257.219,E2 31257.219} C_VEL
LIN {X 0,Y 690.988,Z 1091.056,A -85,B 0,C 180,E1 31255.45,E2 31255.45} C_VEL
LIN {X 0,Y 690.203,Z 1109.257,A -85,B 0,C 180,E1 31253.505,E2 31253.505} C_VEL
LIN {X 0,Y 689.622,Z 1123.693,A -85,B 0,C 180,E1 31251.787,E2 31251.787} C_VEL
LIN {X 0,Y 689.108,Z 1138.964,A -85,B 0,C 180,E1 31249.759,E2 31249.759} C_VEL
LIN {X 0,Y 688.692,Z 1152.675,A -85,B 0,C 180,E1 31247.663,E2 31247.663} C_VEL
LIN {X 0,Y 688.423,Z 1163.15,A -85,B 0,C 180,E1 31245.845,E2 31245.845} C_VEL
LIN {X 0,Y 688.217,Z 1172.777,A -85,B 0,C 180,E1 31243.946,E2 31243.946} C_VEL
LIN {X 0,Y 688.063,Z 1182.005,A -85,B 0,C 180,E1 31241.822,E2 31241.822} C_VEL
LIN {X 0,Y 687.982,Z 1189.819,A -85,B 0,C 180,E1 31239.62,E2 31239.62} C_VEL
LIN {X 0,Y 687.938,Z 1195.972,A -85,B 0,C 180,E1 31237.431,E2 31237.431} C_VEL
LIN {X 0,Y 687.923,Z 1200.64,A -85,B 0,C 180,E1 31235.169,E2 31235.169} C_VEL
LIN {X 0,Y 687.918,Z 1203.517,A -85,B 0,C 180,E1 31232.998,E2 31232.998} C_VEL
LIN {X 0,Y 687.907,Z 1204.777,A -85,B 0,C 180,E1 31230.915,E2 31230.915} C_VEL
LIN {X 0,Y 687.907,Z 1204.777,A -85,B 0,C 180,E1 31229.083,E2 31229.083} C_VEL
LIN {X 0,Y 687.918,Z 1203.436,A -85,B 0,C 180,E1 31226.916,E2 31226.916} C_VEL
LIN {X 0,Y 687.92,Z 1200.489,A -85,B 0,C 180,E1 31224.745,E2 31224.745} C_VEL
LIN {X 0,Y 687.937,Z 1195.772,A -85,B 0,C 180,E1 31222.483,E2 31222.483} C_VEL
LIN {X 0,Y 687.984,Z 1189.544,A -85,B 0,C 180,E1 31220.293,E2 31220.293} C_VEL
LIN {X 0,Y 688.063,Z 1181.997,A -85,B 0,C 180,E1 31218.175,E2 31218.175} C_VEL
LIN {X 0,Y 688.218,Z 1172.725,A -85,B 0,C 180,E1 31216.043,E2 31216.043} C_VEL
LIN {X 0,Y 688.422,Z 1163.139,A -85,B 0,C 180,E1 31214.153,E2 31214.153} C_VEL
LIN {X 0,Y 688.728,Z 1151.617,A -85,B 0,C 180,E1 31212.161,E2 31212.161} C_VEL
LIN {X 0,Y 689.197,Z 1136.394,A -85,B 0,C 180,E1 31209.888,E2 31209.888} C_VEL
LIN {X 0,Y 689.678,Z 1122.255,A -85,B 0,C 180,E1 31208.034,E2 31208.034} C_VEL
LIN {X 0,Y 690.309,Z 1106.367,A -85,B 0,C 180,E1 31206.163,E2 31206.163} C_VEL
LIN {X 0,Y 691.15,Z 1087.792,A -85,B 0,C 180,E1 31204.231,E2 31204.231} C_VEL
LIN {X 0,Y 691.982,Z 1069.496,A -85,B 0,C 180,E1 31202.525,E2 31202.525} C_VEL
LIN {X 0,Y 693.12,Z 1047.108,A -85,B 0,C 180,E1 31200.675,E2 31200.675} C_VEL
LIN {X 0,Y 694.195,Z 1025.613,A -85,B 0,C 180,E1 31199.103,E2 31199.103} C_VEL
LIN {X 0,Y 695.442,Z 1001.049,A -85,B 0,C 180,E1 31197.519,E2 31197.519} C_VEL
LIN {X 0,Y 696.573,Z 978.574,A -85,B 0,C 180,E1 31196.253,E2 31196.253} C_VEL
LIN {X 0,Y 697.577,Z 957.719,A -85,B 0,C 180,E1 31195.215,E2 31195.215} C_VEL
LIN {X 0,Y 698.713,Z 932.497,A -85,B 0,C 180,E1 31194.12,E2 31194.12} C_VEL
LIN {X 0,Y 699.744,Z 906.343,A -85,B 0,C 180,E1 31193.17,E2 31193.17} C_VEL
LIN {X 0,Y 700.657,Z 881.91,A -85,B 0,C 180,E1 31192.43,E2 31192.43} C_VEL
LIN {X 0,Y 701.434,Z 855.492,A -85,B 0,C 180,E1 31191.797,E2 31191.797} C_VEL
LIN {X 0,Y 702.054,Z 828.58,A -85,B 0,C 180,E1 31191.317,E2 31191.317} C_VEL
LIN {X 0,Y 704.199,Z 607.109,A -85,B 0,C 180,E1 31188.542,E2 31188.542} C_VEL
LIN {X 0,Y 706.198,Z 404.123,A -85,B 0,C 180,E1 31185.934,E2 31185.934} C_VEL
LIN {X 0,Y 706.612,Z 350.634,A -85,B 0,C 180,E1 31185.221,E2 31185.221} C_VEL
LIN {X 0,Y 706.301,Z 346.039,A -85,B 0,C 180,E1 31185.131,E2 31185.131} C_VEL
LIN {X 0,Y 697.293,Z 332.658,A -85,B 0,C 180,E1 31184.094,E2 31184.094} C_VEL
LIN {X 0,Y 695.54,Z 329.736,A -85,B 0,C 180,E1 31183.867,E2 31183.867} C_VEL
LIN {X 0,Y 697.251,Z 330.241,A -85,B 0,C 180,E1 31183.732,E2 31183.732} C_VEL
LIN {X 0,Y 700.072,Z 332.068,A -85,B 0,C 180,E1 31183.454,E2 31183.454} C_VEL
LIN {X 0,Y 702.496,Z 334.831,A -85,B 0,C 180,E1 31183.069,E2 31183.069} C_VEL
LIN {X 0,Y 703.929,Z 336.353,A -85,B 0,C 180,E1 31182.626,E2 31182.626} C_VEL
LIN {X 0,Y 704.153,Z 336.862,A -85,B 0,C 180,E1 31182.085,E2 31182.085} C_VEL
LIN {X 0,Y 702.881,Z 336.169,A -85,B 0,C 180,E1 31181.559,E2 31181.559} C_VEL
LIN {X 0,Y 700.46,Z 334.224,A -85,B 0,C 180,E1 31181.093,E2 31181.093} C_VEL
LIN {X 0,Y 696.424,Z 330.128,A -85,B 0,C 180,E1 31180.599,E2 31180.599} C_VEL
LIN {X 0,Y 693.204,Z 326.671,A -85,B 0,C 180,E1 31180.229,E2 31180.229} C_VEL
LIN {X 0,Y 691.592,Z 323.878,A -85,B 0,C 180,E1 31180.017,E2 31180.017} C_VEL
LIN {X 0,Y 689.235,Z 321.105,A -85,B 0,C 180,E1 31179.734,E2 31179.734} C_VEL
LIN {X 0,Y 688.425,Z 318.467,A -85,B 0,C 180,E1 31179.588,E2 31179.588} C_VEL
LIN {X 0,Y 688.458,Z 318.44,A -85,B 0,C 180,E1 31176.567,E2 31176.567} C_VEL
LIN {X 0,Y 688.449,Z 318.476,A -85,B 0,C 180,E1 31173.598,E2 31173.598} C_VEL
LIN {X 0,Y 688.455,Z 318.453,A -85,B 0,C 180,E1 31170.542,E2 31170.542} C_VEL
LIN {X 0,Y 688.459,Z 318.47,A -85,B 0,C 180,E1 31167.452,E2 31167.452} C_VEL
LIN {X 0,Y 688.462,Z 318.454,A -85,B 0,C 180,E1 31164.36,E2 31164.36} C_VEL
LIN {X 0,Y 688.441,Z 318.475,A -85,B 0,C 180,E1 31161.181,E2 31161.181} C_VEL
LIN {X 0,Y 688.467,Z 318.472,A -85,B 0,C 180,E1 31158.195,E2 31158.195} C_VEL
LIN {X 0,Y 688.426,Z 318.478,A -85,B 0,C 180,E1 31155.155,E2 31155.155} C_VEL
LIN {X 0,Y 688.43,Z 318.479,A -85,B 0,C 180,E1 31152.328,E2 31152.328} C_VEL
LIN {X 0,Y 688.466,Z 318.514,A -85,B 0,C 180,E1 31151.817,E2 31151.817} C_VEL
LIN {X 0,Y 689.993,Z 325.116,A -85,B 0,C 180,E1 31151.559,E2 31151.559} C_VEL
LIN {X 0,Y 690.056,Z 400.98,A -85,B 0,C 180,E1 31148.961,E2 31148.961} C_VEL
LIN {X 0,Y 690.472,Z 486.27,A -85,B 0,C 180,E1 31145.901,E2 31145.901} C_VEL
LIN {X 0,Y 690.674,Z 549.272,A -85,B 0,C 180,E1 31143.569,E2 31143.569} C_VEL
LIN {X 0,Y 690.545,Z 620.836,A -85,B 0,C 180,E1 31140.871,E2 31140.871} C_VEL
LIN {X 0,Y 690.117,Z 699.98,A -85,B 0,C 180,E1 31137.841,E2 31137.841} C_VEL
LIN {X 0,Y 689.562,Z 777.262,A -85,B 0,C 180,E1 31134.842,E2 31134.842} C_VEL
LIN {X 0,Y 689.144,Z 838.775,A -85,B 0,C 180,E1 31132.463,E2 31132.463} C_VEL
LIN {X 0,Y 688.943,Z 953.924,A -85,B 0,C 180,E1 31131.245,E2 31131.245} C_VEL
LIN {X 0,Y 688.85,Z 968.225,A -85,B 0,C 180,E1 31130.947,E2 31130.947} C_VEL
LIN {X 0,Y 688.789,Z 976.609,A -85,B 0,C 180,E1 31130.7,E2 31130.7} C_VEL
LIN {X 0,Y 687.743,Z 983.76,A -85,B 0,C 180,E1 31130.461,E2 31130.461} C_VEL
LIN {X 0,Y 683.2,Z 996.313,A -85,B 0,C 180,E1 31129.975,E2 31129.975} C_VEL
LIN {X 0,Y 680.958,Z 1003.793,A -85,B 0,C 180,E1 31129.604,E2 31129.604} C_VEL
LIN {X 0,Y 680.583,Z 1007.294,A -85,B 0,C 180,E1 31129.389,E2 31129.389} C_VEL
LIN {X 0,Y 680.456,Z 1017.623,A -85,B 0,C 180,E1 31128.644,E2 31128.644} C_VEL
LIN {X 0,Y 680.298,Z 1028.082,A -85,B 0,C 180,E1 31127.695,E2 31127.695} C_VEL
LIN {X 0,Y 680.179,Z 1036.883,A -85,B 0,C 180,E1 31126.656,E2 31126.656} C_VEL
LIN {X 0,Y 680.099,Z 1043.415,A -85,B 0,C 180,E1 31125.667,E2 31125.667} C_VEL
LIN {X 0,Y 680.038,Z 1049.339,A -85,B 0,C 180,E1 31124.478,E2 31124.478} C_VEL
LIN {X 0,Y 680.007,Z 1053.138,A -85,B 0,C 180,E1 31123.338,E2 31123.338} C_VEL
LIN {X 0,Y 680.002,Z 1055.312,A -85,B 0,C 180,E1 31122.279,E2 31122.279} C_VEL
LIN {X 0,Y 679.994,Z 1056.299,A -85,B 0,C 180,E1 31121.125,E2 31121.125} C_VEL
LIN {X 0,Y 680,Z 1055.516,A -85,B 0,C 180,E1 31119.784,E2 31119.784} C_VEL
LIN {X 0,Y 680.001,Z 1053.417,A -85,B 0,C 180,E1 31118.703,E2 31118.703} C_VEL
LIN {X 0,Y 680.026,Z 1049.938,A -85,B 0,C 180,E1 31117.615,E2 31117.615} C_VEL
LIN {X 0,Y 680.077,Z 1043.895,A -85,B 0,C 180,E1 31116.345,E2 31116.345} C_VEL
LIN {X 0,Y 680.156,Z 1037.076,A -85,B 0,C 180,E1 31115.301,E2 31115.301} C_VEL
LIN {X 0,Y 680.263,Z 1028.708,A -85,B 0,C 180,E1 31114.303,E2 31114.303} C_VEL
LIN {X 0,Y 680.411,Z 1018.717,A -85,B 0,C 180,E1 31113.371,E2 31113.371} C_VEL
LIN {X 0,Y 680.557,Z 1007.536,A -85,B 0,C 180,E1 31112.55,E2 31112.55} C_VEL
LIN {X 0,Y 680.728,Z 994.386,A -85,B 0,C 180,E1 31111.801,E2 31111.801} C_VEL
LIN {X 0,Y 680.883,Z 980.186,A -85,B 0,C 180,E1 31111.205,E2 31111.205} C_VEL
LIN {X 0,Y 681.004,Z 966.053,A -85,B 0,C 180,E1 31110.785,E2 31110.785} C_VEL
LIN {X 0,Y 681.075,Z 951.064,A -85,B 0,C 180,E1 31110.505,E2 31110.505} C_VEL
LIN {X 0,Y 681.271,Z 837.833,A -85,B 0,C 180,E1 31109.286,E2 31109.286} C_VEL
LIN {X 0,Y 681.933,Z 759.602,A -85,B 0,C 180,E1 31106.204,E2 31106.204} C_VEL
LIN {X 0,Y 682.615,Z 679.459,A -85,B 0,C 180,E1 31103.063,E2 31103.063} C_VEL
LIN {X 0,Y 683.218,Z 602.839,A -85,B 0,C 180,E1 31100.053,E2 31100.053} C_VEL
LIN {X 0,Y 683.692,Z 527.973,A -85,B 0,C 180,E1 31097.114,E2 31097.114} C_VEL
LIN {X 0,Y 684.043,Z 463.131,A -85,B 0,C 180,E1 31094.546,E2 31094.546} C_VEL
LIN {X 0,Y 685.265,Z 464.994,A -85,B 0,C 180,E1 31094.418,E2 31094.418} C_VEL
LIN {X 0,Y 687.04,Z 465.118,A -85,B 0,C 180,E1 31094.271,E2 31094.271} C_VEL
LIN {X 0,Y 689.822,Z 462.97,A -85,B 0,C 180,E1 31094.077,E2 31094.077} C_VEL
LIN {X 0,Y 693.379,Z 457.616,A -85,B 0,C 180,E1 31093.868,E2 31093.868} C_VEL
LIN {X 0,Y 693.829,Z 457.093,A -85,B 0,C 180,E1 31093.839,E2 31093.839} C_VEL
LIN {X 0,Y 697.372,Z 455.77,A -85,B 0,C 180,E1 31093.579,E2 31093.579} C_VEL
LIN {X 0,Y 699.525,Z 454.274,A -85,B 0,C 180,E1 31093.431,E2 31093.431} C_VEL
LIN {X 0,Y 697.29,Z 662.951,A -85,B 0,C 180,E1 31090.762,E2 31090.762} C_VEL
LIN {X 0,Y 695.78,Z 799.23,A -85,B 0,C 180,E1 31089.041,E2 31089.041} C_VEL
LIN {X 0,Y 695.094,Z 826.632,A -85,B 0,C 180,E1 31088.546,E2 31088.546} C_VEL
LIN {X 0,Y 694.156,Z 853.69,A -85,B 0,C 180,E1 31087.881,E2 31087.881} C_VEL
LIN {X 0,Y 693.222,Z 876.484,A -85,B 0,C 180,E1 31087.183,E2 31087.183} C_VEL
LIN {X 0,Y 692.145,Z 900.268,A -85,B 0,C 180,E1 31086.321,E2 31086.321} C_VEL
LIN {X 0,Y 690.859,Z 926.854,A -85,B 0,C 180,E1 31085.172,E2 31085.172} C_VEL
LIN {X 0,Y 689.681,Z 948.65,A -85,B 0,C 180,E1 31084.08,E2 31084.08} C_VEL
LIN {X 0,Y 688.524,Z 969.524,A -85,B 0,C 180,E1 31082.898,E2 31082.898} C_VEL
LIN {X 0,Y 687.16,Z 993.015,A -85,B 0,C 180,E1 31081.395,E2 31081.395} C_VEL
LIN {X 0,Y 685.843,Z 1016.548,A -85,B 0,C 180,E1 31079.667,E2 31079.667} C_VEL
LIN {X 0,Y 684.571,Z 1038.794,A -85,B 0,C 180,E1 31077.819,E2 31077.819} C_VEL
LIN {X 0,Y 683.565,Z 1058.447,A -85,B 0,C 180,E1 31075.967,E2 31075.967} C_VEL
LIN {X 0,Y 682.578,Z 1077.681,A -85,B 0,C 180,E1 31073.924,E2 31073.924} C_VEL
LIN {X 0,Y 681.919,Z 1092.605,A -85,B 0,C 180,E1 31072.139,E2 31072.139} C_VEL
LIN {X 0,Y 681.4,Z 1105.402,A -85,B 0,C 180,E1 31070.442,E2 31070.442} C_VEL
LIN {X 0,Y 680.897,Z 1119.752,A -85,B 0,C 180,E1 31068.317,E2 31068.317} C_VEL
LIN {X 0,Y 680.514,Z 1131.951,A -85,B 0,C 180,E1 31066.211,E2 31066.211} C_VEL
LIN {X 0,Y 680.307,Z 1141.257,A -85,B 0,C 180,E1 31064.383,E2 31064.383} C_VEL
LIN {X 0,Y 680.146,Z 1149.316,A -85,B 0,C 180,E1 31062.568,E2 31062.568} C_VEL
LIN {X 0,Y 680.019,Z 1156.846,A -85,B 0,C 180,E1 31060.592,E2 31060.592} C_VEL
LIN {X 0,Y 679.966,Z 1163.694,A -85,B 0,C 180,E1 31058.372,E2 31058.372} C_VEL
LIN {X 0,Y 679.927,Z 1169.194,A -85,B 0,C 180,E1 31055.994,E2 31055.994} C_VEL
LIN {X 0,Y 679.911,Z 1172.616,A -85,B 0,C 180,E1 31053.795,E2 31053.795} C_VEL
LIN {X 0,Y 679.907,Z 1174.49,A -85,B 0,C 180,E1 31051.686,E2 31051.686} C_VEL
LIN {X 0,Y 679.892,Z 1174.89,A -85,B 0,C 180,E1 31049.411,E2 31049.411} C_VEL
LIN {X 0,Y 679.911,Z 1173.798,A -85,B 0,C 180,E1 31047.219,E2 31047.219} C_VEL
LIN {X 0,Y 679.92,Z 1170.982,A -85,B 0,C 180,E1 31044.939,E2 31044.939} C_VEL
LIN {X 0,Y 679.938,Z 1166.844,A -85,B 0,C 180,E1 31042.821,E2 31042.821} C_VEL
LIN {X 0,Y 679.982,Z 1161.262,A -85,B 0,C 180,E1 31040.693,E2 31040.693} C_VEL
LIN {X 0,Y 680.081,Z 1153.812,A -85,B 0,C 180,E1 31038.467,E2 31038.467} C_VEL
LIN {X 0,Y 680.231,Z 1143.74,A -85,B 0,C 180,E1 31036.052,E2 31036.052} C_VEL
LIN {X 0,Y 680.469,Z 1134.303,A -85,B 0,C 180,E1 31034.14,E2 31034.14} C_VEL
LIN {X 0,Y 680.724,Z 1124.666,A -85,B 0,C 180,E1 31032.42,E2 31032.42} C_VEL
LIN {X 0,Y 681.089,Z 1113.964,A -85,B 0,C 180,E1 31030.713,E2 31030.713} C_VEL
LIN {X 0,Y 681.555,Z 1101.412,A -85,B 0,C 180,E1 31028.917,E2 31028.917} C_VEL
LIN {X 0,Y 682.31,Z 1083.803,A -85,B 0,C 180,E1 31026.694,E2 31026.694} C_VEL
LIN {X 0,Y 683.064,Z 1067.57,A -85,B 0,C 180,E1 31024.882,E2 31024.882} C_VEL
LIN {X 0,Y 684.029,Z 1049.321,A -85,B 0,C 180,E1 31023.056,E2 31023.056} C_VEL
LIN {X 0,Y 685.148,Z 1028.539,A -85,B 0,C 180,E1 31021.212,E2 31021.212} C_VEL
LIN {X 0,Y 686.348,Z 1007.331,A -85,B 0,C 180,E1 31019.539,E2 31019.539} C_VEL
LIN {X 0,Y 687.637,Z 985.104,A -85,B 0,C 180,E1 31017.99,E2 31017.99} C_VEL
LIN {X 0,Y 688.882,Z 963.018,A -85,B 0,C 180,E1 31016.628,E2 31016.628} C_VEL
LIN {X 0,Y 690.269,Z 937.492,A -85,B 0,C 180,E1 31015.251,E2 31015.251} C_VEL
LIN {X 0,Y 691.472,Z 914.648,A -85,B 0,C 180,E1 31014.189,E2 31014.189} C_VEL
LIN {X 0,Y 692.475,Z 893.769,A -85,B 0,C 180,E1 31013.342,E2 31013.342} C_VEL
LIN {X 0,Y 693.484,Z 870.326,A -85,B 0,C 180,E1 31012.524,E2 31012.524} C_VEL
LIN {X 0,Y 694.547,Z 843.172,A -85,B 0,C 180,E1 31011.749,E2 31011.749} C_VEL
LIN {X 0,Y 695.328,Z 817.395,A -85,B 0,C 180,E1 31011.181,E2 31011.181} C_VEL
LIN {X 0,Y 695.887,Z 793.379,A -85,B 0,C 180,E1 31010.785,E2 31010.785} C_VEL
LIN {X 0,Y 698.303,Z 567.863,A -85,B 0,C 180,E1 31007.943,E2 31007.943} C_VEL
LIN {X 0,Y 700.649,Z 357.273,A -85,B 0,C 180,E1 31005.21,E2 31005.21} C_VEL
LIN {X 0,Y 700.624,Z 349.985,A -85,B 0,C 180,E1 31005.105,E2 31005.105} C_VEL
LIN {X 0,Y 686.456,Z 329.06,A -85,B 0,C 180,E1 31003.607,E2 31003.607} C_VEL
LIN {X 0,Y 683.087,Z 324.421,A -85,B 0,C 180,E1 31003.24,E2 31003.24} C_VEL
LIN {X 0,Y 681.061,Z 321.553,A -85,B 0,C 180,E1 31003.015,E2 31003.015} C_VEL
LIN {X 0,Y 680.516,Z 319.465,A -85,B 0,C 180,E1 31002.815,E2 31002.815} C_VEL
LIN {X 0,Y 680.525,Z 319.464,A -85,B 0,C 180,E1 30999.728,E2 30999.728} C_VEL
LIN {X 0,Y 680.512,Z 319.461,A -85,B 0,C 180,E1 30996.658,E2 30996.658} C_VEL
LIN {X 0,Y 680.514,Z 319.44,A -85,B 0,C 180,E1 30993.585,E2 30993.585} C_VEL
LIN {X 0,Y 680.502,Z 319.462,A -85,B 0,C 180,E1 30990.655,E2 30990.655} C_VEL
LIN {X 0,Y 680.503,Z 319.462,A -85,B 0,C 180,E1 30987.761,E2 30987.761} C_VEL
LIN {X 0,Y 680.504,Z 319.442,A -85,B 0,C 180,E1 30984.849,E2 30984.849} C_VEL
LIN {X 0,Y 680.502,Z 319.467,A -85,B 0,C 180,E1 30981.914,E2 30981.914} C_VEL
LIN {X 0,Y 680.522,Z 319.456,A -85,B 0,C 180,E1 30978.948,E2 30978.948} C_VEL
LIN {X 0,Y 680.513,Z 319.442,A -85,B 0,C 180,E1 30975.86,E2 30975.86} C_VEL
LIN {X 0,Y 680.527,Z 319.463,A -85,B 0,C 180,E1 30972.819,E2 30972.819} C_VEL
LIN {X 0,Y 680.512,Z 319.452,A -85,B 0,C 180,E1 30969.728,E2 30969.728} C_VEL
LIN {X 0,Y 680.528,Z 319.44,A -85,B 0,C 180,E1 30966.496,E2 30966.496} C_VEL
LIN {X 0,Y 680.496,Z 319.466,A -85,B 0,C 180,E1 30963.538,E2 30963.538} C_VEL
LIN {X 0,Y 680.523,Z 319.452,A -85,B 0,C 180,E1 30960.505,E2 30960.505} C_VEL
LIN {X 0,Y 680.492,Z 319.443,A -85,B 0,C 180,E1 30957.474,E2 30957.474} C_VEL
LIN {X 0,Y 680.529,Z 319.459,A -85,B 0,C 180,E1 30954.52,E2 30954.52} C_VEL
LIN {X 0,Y 680.513,Z 319.464,A -85,B 0,C 180,E1 30951.295,E2 30951.295} C_VEL
LIN {X 0,Y 680.525,Z 319.443,A -85,B 0,C 180,E1 30948.215,E2 30948.215} C_VEL
LIN {X 0,Y 680.538,Z 319.557,A -85,B 0,C 180,E1 30945.362,E2 30945.362} C_VEL
LIN {X 0,Y 681.899,Z 323.071,A -85,B 0,C 180,E1 30944.783,E2 30944.783} C_VEL
LIN {X 0,Y 683.351,Z 324.862,A -85,B 0,C 180,E1 30944.381,E2 30944.381} C_VEL
LIN {X 0,Y 685.166,Z 328.679,A -85,B 0,C 180,E1 30943.728,E2 30943.728} C_VEL
LIN {X 0,Y 686.235,Z 330.375,A -85,B 0,C 180,E1 30943.406,E2 30943.406} C_VEL
LIN {X 0,Y 689.223,Z 336.047,A -85,B 0,C 180,E1 30942.437,E2 30942.437} C_VEL
LIN {X 0,Y 691.795,Z 340.886,A -85,B 0,C 180,E1 30941.634,E2 30941.634} C_VEL
LIN {X 0,Y 696.353,Z 349.324,A -85,B 0,C 180,E1 30940.279,E2 30940.279} C_VEL
LIN {X 0,Y 701.431,Z 359.558,A -85,B 0,C 180,E1 30938.772,E2 30938.772} C_VEL
LIN {X 0,Y 699.643,Z 394.42,A -85,B 0,C 180,E1 30936.054,E2 30936.054} C_VEL
LIN {X 0,Y 697.879,Z 430.869,A -85,B 0,C 180,E1 30933.355,E2 30933.355} C_VEL
LIN {X 0,Y 696.134,Z 469.419,A -85,B 0,C 180,E1 30930.63,E2 30930.63} C_VEL
LIN {X 0,Y 694.382,Z 511.105,A -85,B 0,C 180,E1 30927.806,E2 30927.806} C_VEL
LIN {X 0,Y 693.497,Z 544.565,A -85,B 0,C 180,E1 30925.584,E2 30925.584} C_VEL
LIN {X 0,Y 694.866,Z 556.996,A -85,B 0,C 180,E1 30924.657,E2 30924.657} C_VEL
LIN {X 0,Y 697.818,Z 567.361,A -85,B 0,C 180,E1 30923.773,E2 30923.773} C_VEL
LIN {X 0,Y 702.04,Z 575.705,A -85,B 0,C 180,E1 30922.953,E2 30922.953} C_VEL
LIN {X 0,Y 707.501,Z 582.569,A -85,B 0,C 180,E1 30922.167,E2 30922.167} C_VEL
LIN {X 0,Y 714.463,Z 588.316,A -85,B 0,C 180,E1 30921.378,E2 30921.378} C_VEL
LIN {X 0,Y 720.15,Z 591.456,A -85,B 0,C 180,E1 30920.821,E2 30920.821} C_VEL
LIN {X 0,Y 723.311,Z 592.352,A -85,B 0,C 180,E1 30920.411,E2 30920.411} C_VEL
LIN {X 0,Y 725.686,Z 592.099,A -85,B 0,C 180,E1 30919.95,E2 30919.95} C_VEL
LIN {X 0,Y 726.889,Z 590.884,A -85,B 0,C 180,E1 30919.513,E2 30919.513} C_VEL
LIN {X 0,Y 727.022,Z 588.375,A -85,B 0,C 180,E1 30919.027,E2 30919.027} C_VEL
LIN {X 0,Y 725.737,Z 584.822,A -85,B 0,C 180,E1 30918.581,E2 30918.581} C_VEL
LIN {X 0,Y 723.095,Z 580.403,A -85,B 0,C 180,E1 30918.214,E2 30918.214} C_VEL
LIN {X 0,Y 716.431,Z 570.557,A -85,B 0,C 180,E1 30917.718,E2 30917.718} C_VEL
LIN {X 0,Y 710.671,Z 559.185,A -85,B 0,C 180,E1 30917.294,E2 30917.294} C_VEL
LIN {X 0,Y 706.137,Z 546.636,A -85,B 0,C 180,E1 30916.954,E2 30916.954} C_VEL
LIN {X 0,Y 702.81,Z 532.875,A -85,B 0,C 180,E1 30916.7,E2 30916.7} C_VEL
LIN {X 0,Y 700.71,Z 517.573,A -85,B 0,C 180,E1 30916.538,E2 30916.538} C_VEL
LIN {X 0,Y 699.899,Z 500.175,A -85,B 0,C 180,E1 30916.475,E2 30916.475} C_VEL
LIN {X 0,Y 699.859,Z 348.098,A -85,B 0,C 180,E1 30916.472,E2 30916.472} C_VEL
LIN {X 0,Y 696.604,Z 349.214,A -85,B 0,C 180,E1 30916.217,E2 30916.217} C_VEL
LIN {X 0,Y 694.082,Z 348.418,A -85,B 0,C 180,E1 30916.017,E2 30916.017} C_VEL
LIN {X 0,Y 693.983,Z 348.451,A -85,B 0,C 180,E1 30915.983,E2 30915.983} C_VEL
LIN {X 0,Y 695.376,Z 351.312,A -85,B 0,C 180,E1 30915.696,E2 30915.696} C_VEL
LIN {X 0,Y 700.83,Z 372.697,A -85,B 0,C 180,E1 30914.936,E2 30914.936} C_VEL
LIN {X 0,Y 698.465,Z 582.203,A -85,B 0,C 180,E1 30912.213,E2 30912.213} C_VEL
LIN {X 0,Y 696.15,Z 805.411,A -85,B 0,C 180,E1 30909.401,E2 30909.401} C_VEL
LIN {X 0,Y 695.631,Z 836.747,A -85,B 0,C 180,E1 30908.969,E2 30908.969} C_VEL
LIN {X 0,Y 694.854,Z 864.001,A -85,B 0,C 180,E1 30908.428,E2 30908.428} C_VEL
LIN {X 0,Y 693.921,Z 889.916,A -85,B 0,C 180,E1 30907.75,E2 30907.75} C_VEL
LIN {X 0,Y 692.794,Z 917.571,A -85,B 0,C 180,E1 30906.845,E2 30906.845} C_VEL
LIN {X 0,Y 691.688,Z 940.713,A -85,B 0,C 180,E1 30905.936,E2 30905.936} C_VEL
LIN {X 0,Y 690.572,Z 962.169,A -85,B 0,C 180,E1 30904.963,E2 30904.963} C_VEL
LIN {X 0,Y 689.237,Z 986.499,A -85,B 0,C 180,E1 30903.702,E2 30903.702} C_VEL
LIN {X 0,Y 687.892,Z 1010.105,A -85,B 0,C 180,E1 30902.287,E2 30902.287} C_VEL
LIN {X 0,Y 686.765,Z 1030.286,A -85,B 0,C 180,E1 30900.925,E2 30900.925} C_VEL
LIN {X 0,Y 685.532,Z 1052.011,A -85,B 0,C 180,E1 30899.282,E2 30899.282} C_VEL
LIN {X 0,Y 684.337,Z 1073.364,A -85,B 0,C 180,E1 30897.449,E2 30897.449} C_VEL
LIN {X 0,Y 683.328,Z 1092.871,A -85,B 0,C 180,E1 30895.572,E2 30895.572} C_VEL
LIN {X 0,Y 682.469,Z 1110.287,A -85,B 0,C 180,E1 30893.667,E2 30893.667} C_VEL
LIN {X 0,Y 681.809,Z 1125.116,A -85,B 0,C 180,E1 30891.868,E2 30891.868} C_VEL
LIN {X 0,Y 681.177,Z 1141.381,A -85,B 0,C 180,E1 30889.641,E2 30889.641} C_VEL
LIN {X 0,Y 680.746,Z 1154.396,A -85,B 0,C 180,E1 30887.586,E2 30887.586} C_VEL
LIN {X 0,Y 680.45,Z 1165.014,A -85,B 0,C 180,E1 30885.686,E2 30885.686} C_VEL
LIN {X 0,Y 680.214,Z 1175.933,A -85,B 0,C 180,E1 30883.429,E2 30883.429} C_VEL
LIN {X 0,Y 680.039,Z 1185.224,A -85,B 0,C 180,E1 30881.104,E2 30881.104} C_VEL
LIN {X 0,Y 679.966,Z 1192.388,A -85,B 0,C 180,E1 30878.881,E2 30878.881} C_VEL
LIN {X 0,Y 679.928,Z 1197.914,A -85,B 0,C 180,E1 30876.67,E2 30876.67} C_VEL
LIN {X 0,Y 679.916,Z 1201.925,A -85,B 0,C 180,E1 30874.381,E2 30874.381} C_VEL
LIN {X 0,Y 679.912,Z 1204.209,A -85,B 0,C 180,E1 30872.19,E2 30872.19} C_VEL
LIN {X 0,Y 679.903,Z 1204.969,A -85,B 0,C 180,E1 30869.83,E2 30869.83} C_VEL
LIN {X 0,Y 679.907,Z 1204.039,A -85,B 0,C 180,E1 30867.555,E2 30867.555} C_VEL
LIN {X 0,Y 679.91,Z 1201.544,A -85,B 0,C 180,E1 30865.36,E2 30865.36} C_VEL
LIN {X 0,Y 679.927,Z 1197.531,A -85,B 0,C 180,E1 30863.158,E2 30863.158} C_VEL
LIN {X 0,Y 679.974,Z 1191.651,A -85,B 0,C 180,E1 30860.861,E2 30860.861} C_VEL
LIN {X 0,Y 680.067,Z 1184.274,A -85,B 0,C 180,E1 30858.637,E2 30858.637} C_VEL
LIN {X 0,Y 680.237,Z 1174.371,A -85,B 0,C 180,E1 30856.223,E2 30856.223} C_VEL
LIN {X 0,Y 680.474,Z 1164.072,A -85,B 0,C 180,E1 30854.138,E2 30854.138} C_VEL
LIN {X 0,Y 680.77,Z 1153.71,A -85,B 0,C 180,E1 30852.299,E2 30852.299} C_VEL
LIN {X 0,Y 681.232,Z 1140.159,A -85,B 0,C 180,E1 30850.18,E2 30850.18} C_VEL
LIN {X 0,Y 681.837,Z 1124.389,A -85,B 0,C 180,E1 30848.04,E2 30848.04} C_VEL
LIN {X 0,Y 682.479,Z 1110.025,A -85,B 0,C 180,E1 30846.303,E2 30846.303} C_VEL
LIN {X 0,Y 683.354,Z 1092.392,A -85,B 0,C 180,E1 30844.381,E2 30844.381} C_VEL
LIN {X 0,Y 684.339,Z 1073.339,A -85,B 0,C 180,E1 30842.549,E2 30842.549} C_VEL
LIN {X 0,Y 685.532,Z 1052.011,A -85,B 0,C 180,E1 30840.718,E2 30840.718} C_VEL
LIN {X 0,Y 686.766,Z 1030.254,A -85,B 0,C 180,E1 30839.072,E2 30839.072} C_VEL
LIN {X 0,Y 687.895,Z 1010.07,A -85,B 0,C 180,E1 30837.711,E2 30837.711} C_VEL
LIN {X 0,Y 689.295,Z 985.61,A -85,B 0,C 180,E1 30836.249,E2 30836.249} C_VEL
LIN {X 0,Y 690.598,Z 961.701,A -85,B 0,C 180,E1 30835.015,E2 30835.015} C_VEL
LIN {X 0,Y 691.707,Z 940.329,A -85,B 0,C 180,E1 30834.048,E2 30834.048} C_VEL
LIN {X 0,Y 692.826,Z 916.843,A -85,B 0,C 180,E1 30833.129,E2 30833.129} C_VEL
LIN {X 0,Y 693.946,Z 889.084,A -85,B 0,C 180,E1 30832.225,E2 30832.225} C_VEL
LIN {X 0,Y 694.879,Z 863.158,A -85,B 0,C 180,E1 30831.554,E2 30831.554} C_VEL
LIN {X 0,Y 695.658,Z 835.759,A -85,B 0,C 180,E1 30831.014,E2 30831.014} C_VEL
LIN {X 0,Y 696.191,Z 801.491,A -85,B 0,C 180,E1 30830.55,E2 30830.55} C_VEL
LIN {X 0,Y 698.517,Z 577.588,A -85,B 0,C 180,E1 30827.728,E2 30827.728} C_VEL
LIN {X 0,Y 700.944,Z 364.64,A -85,B 0,C 180,E1 30824.959,E2 30824.959} C_VEL
LIN {X 0,Y 700.823,Z 350.15,A -85,B 0,C 180,E1 30824.742,E2 30824.742} C_VEL
LIN {X 0,Y 694.105,Z 340.127,A -85,B 0,C 180,E1 30823.981,E2 30823.981} C_VEL
LIN {X 0,Y 696.599,Z 339.794,A -85,B 0,C 180,E1 30823.78,E2 30823.78} C_VEL
LIN {X 0,Y 697.608,Z 339.171,A -85,B 0,C 180,E1 30823.688,E2 30823.688} C_VEL
LIN {X 0,Y 700.646,Z 342.111,A -85,B 0,C 180,E1 30823.296,E2 30823.296} C_VEL
LIN {X 0,Y 702.616,Z 343.981,A -85,B 0,C 180,E1 30822.81,E2 30822.81} C_VEL
LIN {X 0,Y 703.128,Z 344.752,A -85,B 0,C 180,E1 30822.271,E2 30822.271} C_VEL
LIN {X 0,Y 702.059,Z 344.44,A -85,B 0,C 180,E1 30821.729,E2 30821.729} C_VEL
LIN {X 0,Y 699.761,Z 343.111,A -85,B 0,C 180,E1 30821.257,E2 30821.257} C_VEL
LIN {X 0,Y 696.152,Z 340.336,A -85,B 0,C 180,E1 30820.808,E2 30820.808} C_VEL
LIN {X 0,Y 691.835,Z 336.18,A -85,B 0,C 180,E1 30820.325,E2 30820.325} C_VEL
LIN {X 0,Y 688.356,Z 331.775,A -85,B 0,C 180,E1 30819.904,E2 30819.904} C_VEL
LIN {X 0,Y 686.753,Z 329.592,A -85,B 0,C 180,E1 30819.703,E2 30819.703} C_VEL
LIN {X 0,Y 684.183,Z 325.572,A -85,B 0,C 180,E1 30819.366,E2 30819.366} C_VEL
LIN {X 0,Y 681.251,Z 321.945,A -85,B 0,C 180,E1 30818.998,E2 30818.998} C_VEL
LIN {X 0,Y 680.531,Z 319.464,A -85,B 0,C 180,E1 30818.856,E2 30818.856} C_VEL
LIN {X 0,Y 680.483,Z 319.437,A -85,B 0,C 180,E1 30815.79,E2 30815.79} C_VEL
LIN {X 0,Y 680.49,Z 319.457,A -85,B 0,C 180,E1 30812.964,E2 30812.964} C_VEL
LIN {X 0,Y 680.527,Z 319.449,A -85,B 0,C 180,E1 30809.971,E2 30809.971} C_VEL
LIN {X 0,Y 680.504,Z 319.454,A -85,B 0,C 180,E1 30807.002,E2 30807.002} C_VEL
LIN {X 0,Y 680.52,Z 319.453,A -85,B 0,C 180,E1 30803.74,E2 30803.74} C_VEL
LIN {X 0,Y 680.519,Z 319.456,A -85,B 0,C 180,E1 30800.739,E2 30800.739} C_VEL
LIN {X 0,Y 680.51,Z 319.46,A -85,B 0,C 180,E1 30797.619,E2 30797.619} C_VEL
LIN {X 0,Y 680.51,Z 319.467,A -85,B 0,C 180,E1 30794.639,E2 30794.639} C_VEL
LIN {X 0,Y 680.534,Z 319.59,A -85,B 0,C 180,E1 30791.967,E2 30791.967} C_VEL
LIN {X 0,Y 682.26,Z 326.544,A -85,B 0,C 180,E1 30791.695,E2 30791.695} C_VEL
LIN {X 0,Y 682.321,Z 400.88,A -85,B 0,C 180,E1 30789.149,E2 30789.149} C_VEL
LIN {X 0,Y 682.718,Z 483.795,A -85,B 0,C 180,E1 30786.18,E2 30786.18} C_VEL
LIN {X 0,Y 682.957,Z 554.46,A -85,B 0,C 180,E1 30783.567,E2 30783.567} C_VEL
LIN {X 0,Y 682.725,Z 634.015,A -85,B 0,C 180,E1 30780.545,E2 30780.545} C_VEL
LIN {X 0,Y 682.341,Z 703.053,A -85,B 0,C 180,E1 30777.901,E2 30777.901} C_VEL
LIN {X 0,Y 681.757,Z 780.997,A -85,B 0,C 180,E1 30774.867,E2 30774.867} C_VEL
LIN {X 0,Y 681.331,Z 840.033,A -85,B 0,C 180,E1 30772.578,E2 30772.578} C_VEL
LIN {X 0,Y 681.058,Z 954.834,A -85,B 0,C 180,E1 30771.348,E2 30771.348} C_VEL
LIN {X 0,Y 680.975,Z 969.754,A -85,B 0,C 180,E1 30771.035,E2 30771.035} C_VEL
LIN {X 0,Y 680.859,Z 985.01,A -85,B 0,C 180,E1 30770.533,E2 30770.533} C_VEL
LIN {X 0,Y 680.714,Z 997.971,A -85,B 0,C 180,E1 30769.933,E2 30769.933} C_VEL
LIN {X 0,Y 680.583,Z 1007.294,A -85,B 0,C 180,E1 30769.389,E2 30769.389} C_VEL
LIN {X 0,Y 679.551,Z 1013.42,A -85,B 0,C 180,E1 30768.993,E2 30768.993} C_VEL
